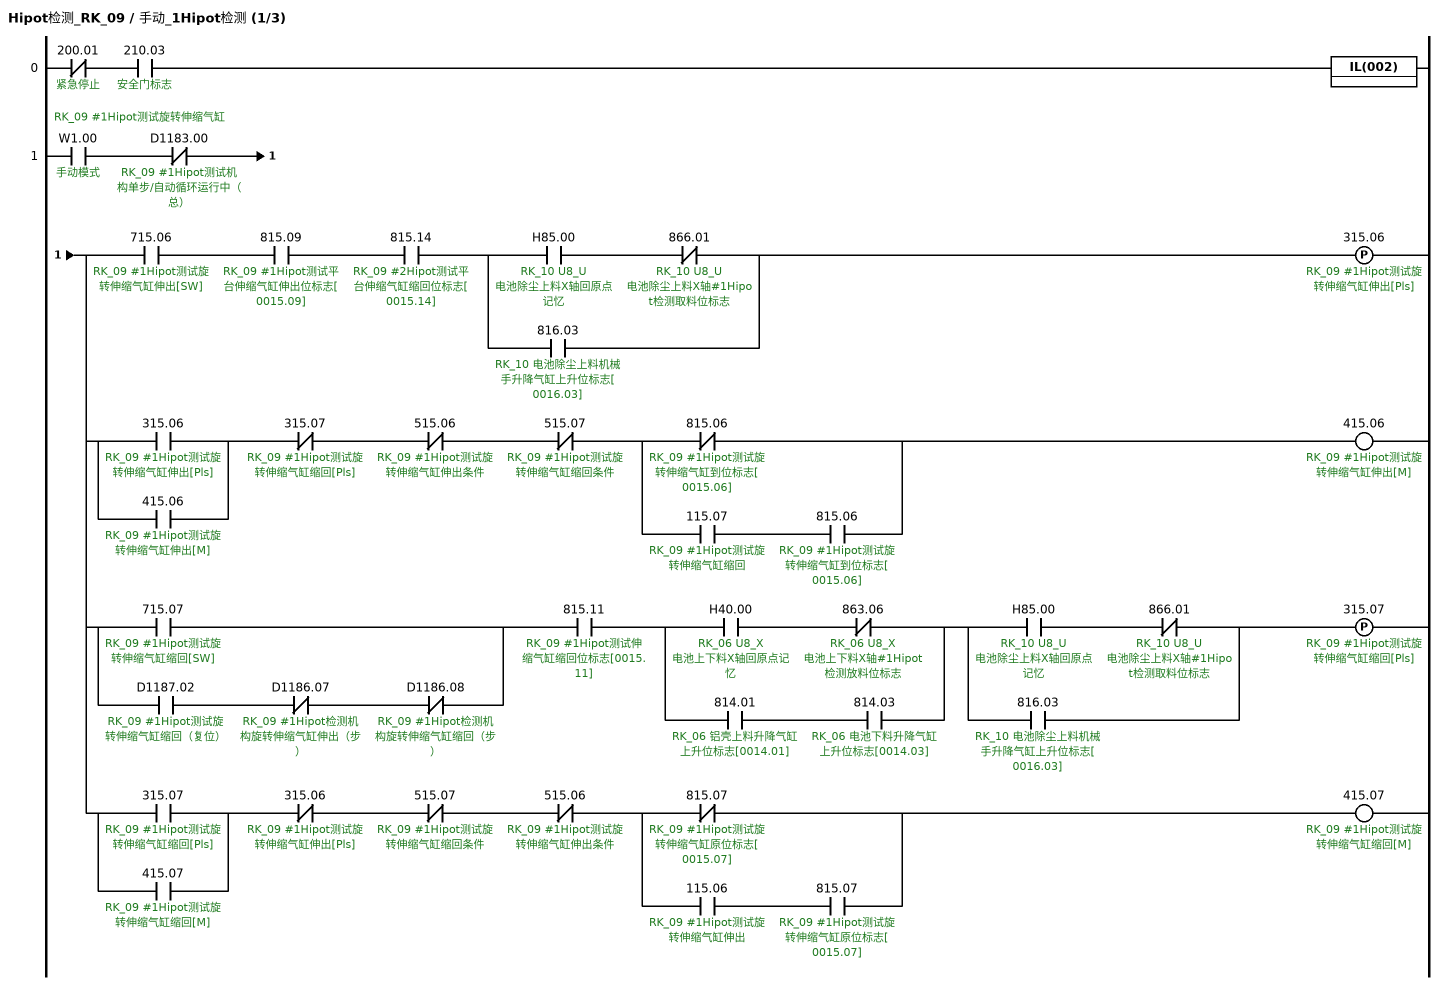
; [picture p648: Hipot检测_RK_09 / 手动_1Hipot检测, rungs 0-1]
; rung 0
LDNOT 200.01  ; 紧急停止
AND 210.03  ; 安全门标志
IL(002)
; rung 1: RK_09 #1Hipot测试旋转伸缩气缸
LD W1.00  ; 手动模式
ANDNOT D1183.00  ; RK_09 #1Hipot测试机构单步/自动循环运行中（总）
OUT TR0
AND 715.06  ; RK_09 #1Hipot测试旋转伸缩气缸伸出[SW]
AND 815.09  ; RK_09 #1Hipot测试平台伸缩气缸伸出位标志[0015.09]
AND 815.14  ; RK_09 #2Hipot测试平台伸缩气缸缩回位标志[0015.14]
LD H85.00  ; RK_10 U8_U 电池除尘上料X轴回原点记忆
ANDNOT 866.01  ; RK_10 U8_U 电池除尘上料X轴#1Hipot检测取料位标志
OR 816.03  ; RK_10 电池除尘上料机械手升降气缸上升位标志[0016.03]
ANDLD
DIFU(013) 315.06  ; RK_09 #1Hipot测试旋转伸缩气缸伸出[Pls]
LD TR0
LD 315.06  ; RK_09 #1Hipot测试旋转伸缩气缸伸出[Pls]
OR 415.06  ; RK_09 #1Hipot测试旋转伸缩气缸伸出[M]
ANDLD
ANDNOT 315.07  ; RK_09 #1Hipot测试旋转伸缩气缸缩回[Pls]
ANDNOT 515.06  ; RK_09 #1Hipot测试旋转伸缩气缸伸出条件
ANDNOT 515.07  ; RK_09 #1Hipot测试旋转伸缩气缸缩回条件
LDNOT 815.06  ; RK_09 #1Hipot测试旋转伸缩气缸到位标志[0015.06]
LD 115.07  ; RK_09 #1Hipot测试旋转伸缩气缸缩回
AND 815.06  ; RK_09 #1Hipot测试旋转伸缩气缸到位标志[0015.06]
ORLD
ANDLD
OUT 415.06  ; RK_09 #1Hipot测试旋转伸缩气缸伸出[M]
LD TR0
LD 715.07  ; RK_09 #1Hipot测试旋转伸缩气缸缩回[SW]
LD D1187.02  ; RK_09 #1Hipot测试旋转伸缩气缸缩回（复位）
ANDNOT D1186.07  ; RK_09 #1Hipot检测机构旋转伸缩气缸伸出（步）
ANDNOT D1186.08  ; RK_09 #1Hipot检测机构旋转伸缩气缸缩回（步）
ORLD
ANDLD
AND 815.11  ; RK_09 #1Hipot测试伸缩气缸缩回位标志[0015.11]
LD H40.00  ; RK_06 U8_X 电池上下料X轴回原点记忆
ANDNOT 863.06  ; RK_06 U8_X 电池上下料X轴#1Hipot检测放料位标志
LD 814.01  ; RK_06 铝壳上料升降气缸上升位标志[0014.01]
AND 814.03  ; RK_06 电池下料升降气缸上升位标志[0014.03]
ORLD
ANDLD
LD H85.00  ; RK_10 U8_U 电池除尘上料X轴回原点记忆
ANDNOT 866.01  ; RK_10 U8_U 电池除尘上料X轴#1Hipot检测取料位标志
OR 816.03  ; RK_10 电池除尘上料机械手升降气缸上升位标志[0016.03]
ANDLD
DIFU(013) 315.07  ; RK_09 #1Hipot测试旋转伸缩气缸缩回[Pls]
LD TR0
LD 315.07  ; RK_09 #1Hipot测试旋转伸缩气缸缩回[Pls]
OR 415.07  ; RK_09 #1Hipot测试旋转伸缩气缸缩回[M]
ANDLD
ANDNOT 315.06  ; RK_09 #1Hipot测试旋转伸缩气缸伸出[Pls]
ANDNOT 515.07  ; RK_09 #1Hipot测试旋转伸缩气缸缩回条件
ANDNOT 515.06  ; RK_09 #1Hipot测试旋转伸缩气缸伸出条件
LDNOT 815.07  ; RK_09 #1Hipot测试旋转伸缩气缸原位标志[0015.07]
LD 115.06  ; RK_09 #1Hipot测试旋转伸缩气缸伸出
AND 815.07  ; RK_09 #1Hipot测试旋转伸缩气缸原位标志[0015.07]
ORLD
ANDLD
OUT 415.07  ; RK_09 #1Hipot测试旋转伸缩气缸缩回[M]

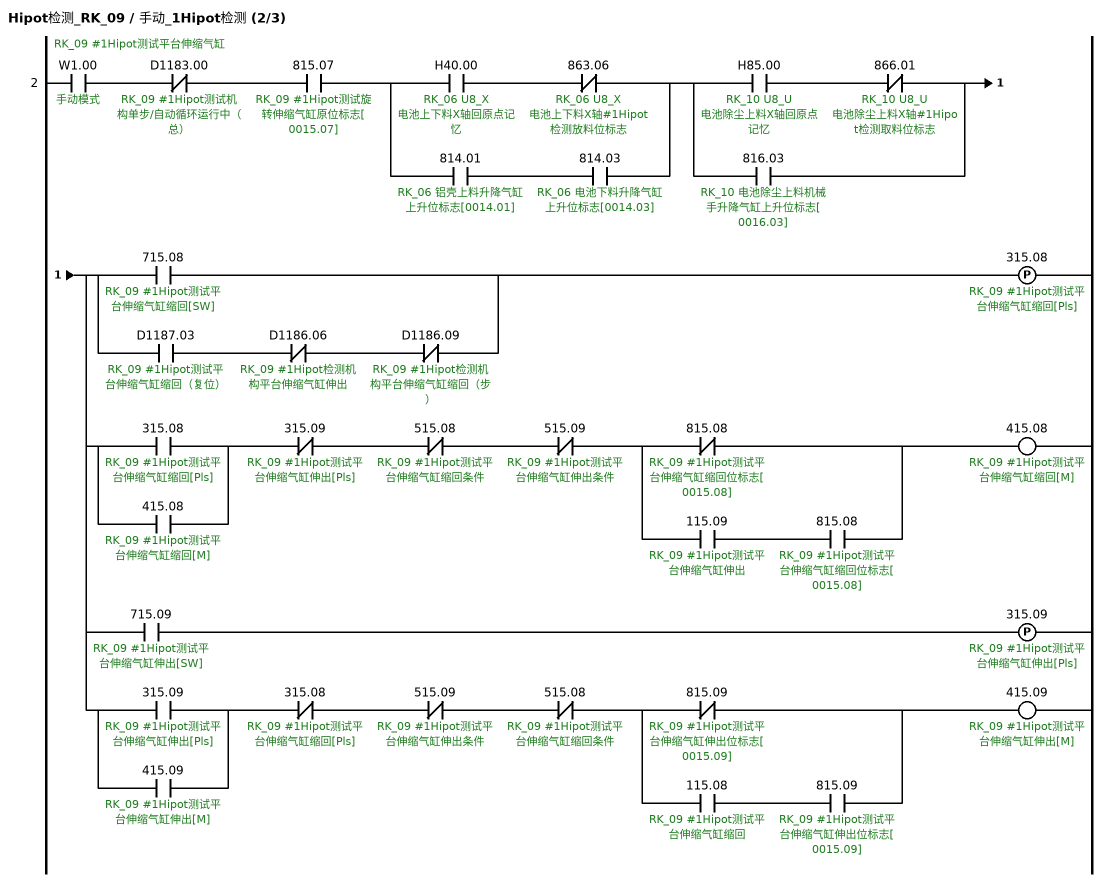
; rung 2: RK_09 #1Hipot测试平台伸缩气缸
LD W1.00  ; 手动模式
ANDNOT D1183.00  ; RK_09 #1Hipot测试机构单步/自动循环运行中（总）
AND 815.07  ; RK_09 #1Hipot测试旋转伸缩气缸原位标志[0015.07]
LD H40.00  ; RK_06 U8_X 电池上下料X轴回原点记忆
ANDNOT 863.06  ; RK_06 U8_X 电池上下料X轴#1Hipot检测放料位标志
LD 814.01  ; RK_06 铝壳上料升降气缸上升位标志[0014.01]
AND 814.03  ; RK_06 电池下料升降气缸上升位标志[0014.03]
ORLD
ANDLD
LD H85.00  ; RK_10 U8_U 电池除尘上料X轴回原点记忆
ANDNOT 866.01  ; RK_10 U8_U 电池除尘上料X轴#1Hipot检测取料位标志
OR 816.03  ; RK_10 电池除尘上料机械手升降气缸上升位标志[0016.03]
ANDLD
OUT TR0
LD 715.08  ; RK_09 #1Hipot测试平台伸缩气缸缩回[SW]
LD D1187.03  ; RK_09 #1Hipot测试平台伸缩气缸缩回（复位）
ANDNOT D1186.06  ; RK_09 #1Hipot检测机构平台伸缩气缸伸出
ANDNOT D1186.09  ; RK_09 #1Hipot检测机构平台伸缩气缸缩回（步）
ORLD
ANDLD
DIFU(013) 315.08  ; RK_09 #1Hipot测试平台伸缩气缸缩回[Pls]
LD TR0
LD 315.08  ; RK_09 #1Hipot测试平台伸缩气缸缩回[Pls]
OR 415.08  ; RK_09 #1Hipot测试平台伸缩气缸缩回[M]
ANDLD
ANDNOT 315.09  ; RK_09 #1Hipot测试平台伸缩气缸伸出[Pls]
ANDNOT 515.08  ; RK_09 #1Hipot测试平台伸缩气缸缩回条件
ANDNOT 515.09  ; RK_09 #1Hipot测试平台伸缩气缸伸出条件
LDNOT 815.08  ; RK_09 #1Hipot测试平台伸缩气缸缩回位标志[0015.08]
LD 115.09  ; RK_09 #1Hipot测试平台伸缩气缸伸出
AND 815.08  ; RK_09 #1Hipot测试平台伸缩气缸缩回位标志[0015.08]
ORLD
ANDLD
OUT 415.08  ; RK_09 #1Hipot测试平台伸缩气缸缩回[M]
LD TR0
AND 715.09  ; RK_09 #1Hipot测试平台伸缩气缸伸出[SW]
DIFU(013) 315.09  ; RK_09 #1Hipot测试平台伸缩气缸伸出[Pls]
LD TR0
LD 315.09  ; RK_09 #1Hipot测试平台伸缩气缸伸出[Pls]
OR 415.09  ; RK_09 #1Hipot测试平台伸缩气缸伸出[M]
ANDLD
ANDNOT 315.08  ; RK_09 #1Hipot测试平台伸缩气缸缩回[Pls]
ANDNOT 515.09  ; RK_09 #1Hipot测试平台伸缩气缸伸出条件
ANDNOT 515.08  ; RK_09 #1Hipot测试平台伸缩气缸缩回条件
LDNOT 815.09  ; RK_09 #1Hipot测试平台伸缩气缸伸出位标志[0015.09]
LD 115.08  ; RK_09 #1Hipot测试平台伸缩气缸缩回
AND 815.09  ; RK_09 #1Hipot测试平台伸缩气缸伸出位标志[0015.09]
ORLD
ANDLD
OUT 415.09  ; RK_09 #1Hipot测试平台伸缩气缸伸出[M]

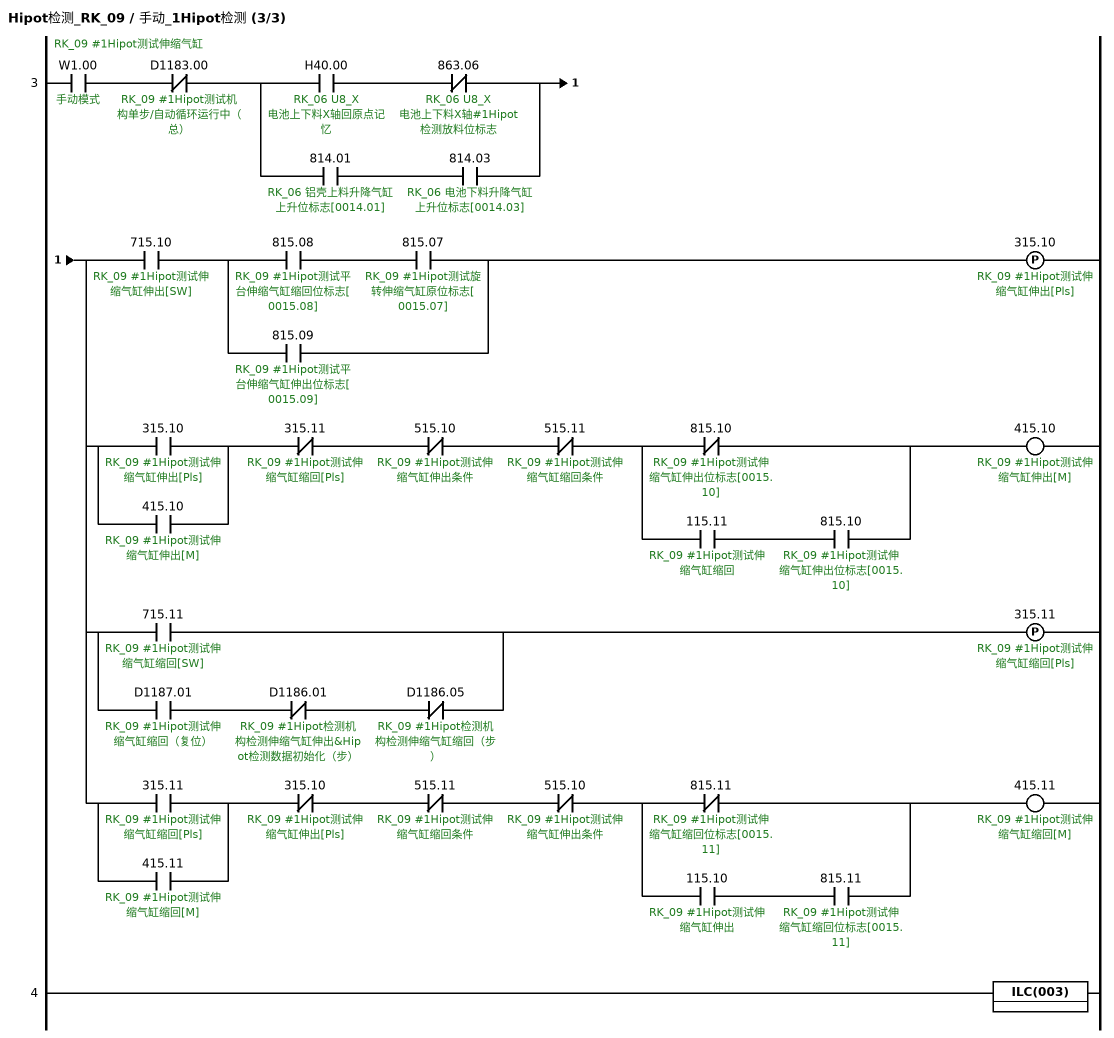
; rung 3: RK_09 #1Hipot测试伸缩气缸
LD W1.00  ; 手动模式
ANDNOT D1183.00  ; RK_09 #1Hipot测试机构单步/自动循环运行中（总）
LD H40.00  ; RK_06 U8_X 电池上下料X轴回原点记忆
ANDNOT 863.06  ; RK_06 U8_X 电池上下料X轴#1Hipot检测放料位标志
LD 814.01  ; RK_06 铝壳上料升降气缸上升位标志[0014.01]
AND 814.03  ; RK_06 电池下料升降气缸上升位标志[0014.03]
ORLD
ANDLD
OUT TR0
AND 715.10  ; RK_09 #1Hipot测试伸缩气缸伸出[SW]
LD 815.08  ; RK_09 #1Hipot测试平台伸缩气缸缩回位标志[0015.08]
AND 815.07  ; RK_09 #1Hipot测试旋转伸缩气缸原位标志[0015.07]
OR 815.09  ; RK_09 #1Hipot测试平台伸缩气缸伸出位标志[0015.09]
ANDLD
DIFU(013) 315.10  ; RK_09 #1Hipot测试伸缩气缸伸出[Pls]
LD TR0
LD 315.10  ; RK_09 #1Hipot测试伸缩气缸伸出[Pls]
OR 415.10  ; RK_09 #1Hipot测试伸缩气缸伸出[M]
ANDLD
ANDNOT 315.11  ; RK_09 #1Hipot测试伸缩气缸缩回[Pls]
ANDNOT 515.10  ; RK_09 #1Hipot测试伸缩气缸伸出条件
ANDNOT 515.11  ; RK_09 #1Hipot测试伸缩气缸缩回条件
LDNOT 815.10  ; RK_09 #1Hipot测试伸缩气缸伸出位标志[0015.10]
LD 115.11  ; RK_09 #1Hipot测试伸缩气缸缩回
AND 815.10  ; RK_09 #1Hipot测试伸缩气缸伸出位标志[0015.10]
ORLD
ANDLD
OUT 415.10  ; RK_09 #1Hipot测试伸缩气缸伸出[M]
LD TR0
LD 715.11  ; RK_09 #1Hipot测试伸缩气缸缩回[SW]
LD D1187.01  ; RK_09 #1Hipot测试伸缩气缸缩回（复位）
ANDNOT D1186.01  ; RK_09 #1Hipot检测机构检测伸缩气缸伸出&Hipot检测数据初始化（步）
ANDNOT D1186.05  ; RK_09 #1Hipot检测机构检测伸缩气缸缩回（步）
ORLD
ANDLD
DIFU(013) 315.11  ; RK_09 #1Hipot测试伸缩气缸缩回[Pls]
LD TR0
LD 315.11  ; RK_09 #1Hipot测试伸缩气缸缩回[Pls]
OR 415.11  ; RK_09 #1Hipot测试伸缩气缸缩回[M]
ANDLD
ANDNOT 315.10  ; RK_09 #1Hipot测试伸缩气缸伸出[Pls]
ANDNOT 515.11  ; RK_09 #1Hipot测试伸缩气缸缩回条件
ANDNOT 515.10  ; RK_09 #1Hipot测试伸缩气缸伸出条件
LDNOT 815.11  ; RK_09 #1Hipot测试伸缩气缸缩回位标志[0015.11]
LD 115.10  ; RK_09 #1Hipot测试伸缩气缸伸出
AND 815.11  ; RK_09 #1Hipot测试伸缩气缸缩回位标志[0015.11]
ORLD
ANDLD
OUT 415.11  ; RK_09 #1Hipot测试伸缩气缸缩回[M]
; rung 4
ILC(003)

### Section 手动_2Hipot检测

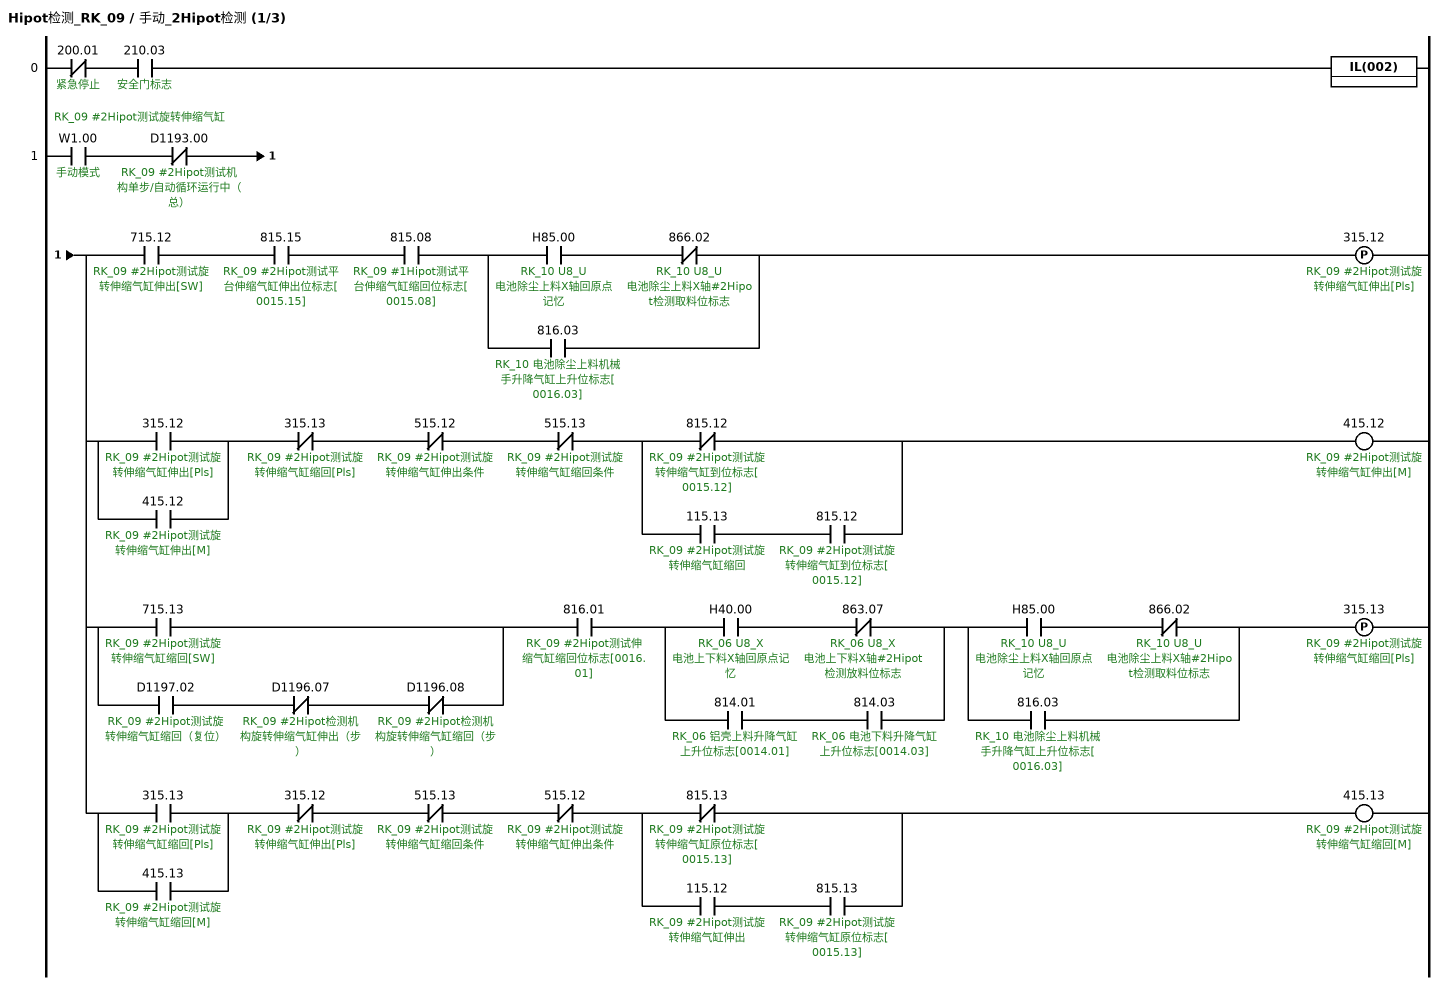
; rung 0
LDNOT 200.01  ; 紧急停止
AND 210.03  ; 安全门标志
IL(002)
; rung 1: RK_09 #2Hipot测试旋转伸缩气缸
LD W1.00  ; 手动模式
ANDNOT D1193.00  ; RK_09 #2Hipot测试机构单步/自动循环运行中（总）
OUT TR0
AND 715.12  ; RK_09 #2Hipot测试旋转伸缩气缸伸出[SW]
AND 815.15  ; RK_09 #2Hipot测试平台伸缩气缸伸出位标志[0015.15]
AND 815.08  ; RK_09 #1Hipot测试平台伸缩气缸缩回位标志[0015.08]
LD H85.00  ; RK_10 U8_U 电池除尘上料X轴回原点记忆
ANDNOT 866.02  ; RK_10 U8_U 电池除尘上料X轴#2Hipot检测取料位标志
OR 816.03  ; RK_10 电池除尘上料机械手升降气缸上升位标志[0016.03]
ANDLD
DIFU(013) 315.12  ; RK_09 #2Hipot测试旋转伸缩气缸伸出[Pls]
LD TR0
LD 315.12  ; RK_09 #2Hipot测试旋转伸缩气缸伸出[Pls]
OR 415.12  ; RK_09 #2Hipot测试旋转伸缩气缸伸出[M]
ANDLD
ANDNOT 315.13  ; RK_09 #2Hipot测试旋转伸缩气缸缩回[Pls]
ANDNOT 515.12  ; RK_09 #2Hipot测试旋转伸缩气缸伸出条件
ANDNOT 515.13  ; RK_09 #2Hipot测试旋转伸缩气缸缩回条件
LDNOT 815.12  ; RK_09 #2Hipot测试旋转伸缩气缸到位标志[0015.12]
LD 115.13  ; RK_09 #2Hipot测试旋转伸缩气缸缩回
AND 815.12  ; RK_09 #2Hipot测试旋转伸缩气缸到位标志[0015.12]
ORLD
ANDLD
OUT 415.12  ; RK_09 #2Hipot测试旋转伸缩气缸伸出[M]
LD TR0
LD 715.13  ; RK_09 #2Hipot测试旋转伸缩气缸缩回[SW]
LD D1197.02  ; RK_09 #2Hipot测试旋转伸缩气缸缩回（复位）
ANDNOT D1196.07  ; RK_09 #2Hipot检测机构旋转伸缩气缸伸出（步）
ANDNOT D1196.08  ; RK_09 #2Hipot检测机构旋转伸缩气缸缩回（步）
ORLD
ANDLD
AND 816.01  ; RK_09 #2Hipot测试伸缩气缸缩回位标志[0016.01]
LD H40.00  ; RK_06 U8_X 电池上下料X轴回原点记忆
ANDNOT 863.07  ; RK_06 U8_X 电池上下料X轴#2Hipot检测放料位标志
LD 814.01  ; RK_06 铝壳上料升降气缸上升位标志[0014.01]
AND 814.03  ; RK_06 电池下料升降气缸上升位标志[0014.03]
ORLD
ANDLD
LD H85.00  ; RK_10 U8_U 电池除尘上料X轴回原点记忆
ANDNOT 866.02  ; RK_10 U8_U 电池除尘上料X轴#2Hipot检测取料位标志
OR 816.03  ; RK_10 电池除尘上料机械手升降气缸上升位标志[0016.03]
ANDLD
DIFU(013) 315.13  ; RK_09 #2Hipot测试旋转伸缩气缸缩回[Pls]
LD TR0
LD 315.13  ; RK_09 #2Hipot测试旋转伸缩气缸缩回[Pls]
OR 415.13  ; RK_09 #2Hipot测试旋转伸缩气缸缩回[M]
ANDLD
ANDNOT 315.12  ; RK_09 #2Hipot测试旋转伸缩气缸伸出[Pls]
ANDNOT 515.13  ; RK_09 #2Hipot测试旋转伸缩气缸缩回条件
ANDNOT 515.12  ; RK_09 #2Hipot测试旋转伸缩气缸伸出条件
LDNOT 815.13  ; RK_09 #2Hipot测试旋转伸缩气缸原位标志[0015.13]
LD 115.12  ; RK_09 #2Hipot测试旋转伸缩气缸伸出
AND 815.13  ; RK_09 #2Hipot测试旋转伸缩气缸原位标志[0015.13]
ORLD
ANDLD
OUT 415.13  ; RK_09 #2Hipot测试旋转伸缩气缸缩回[M]

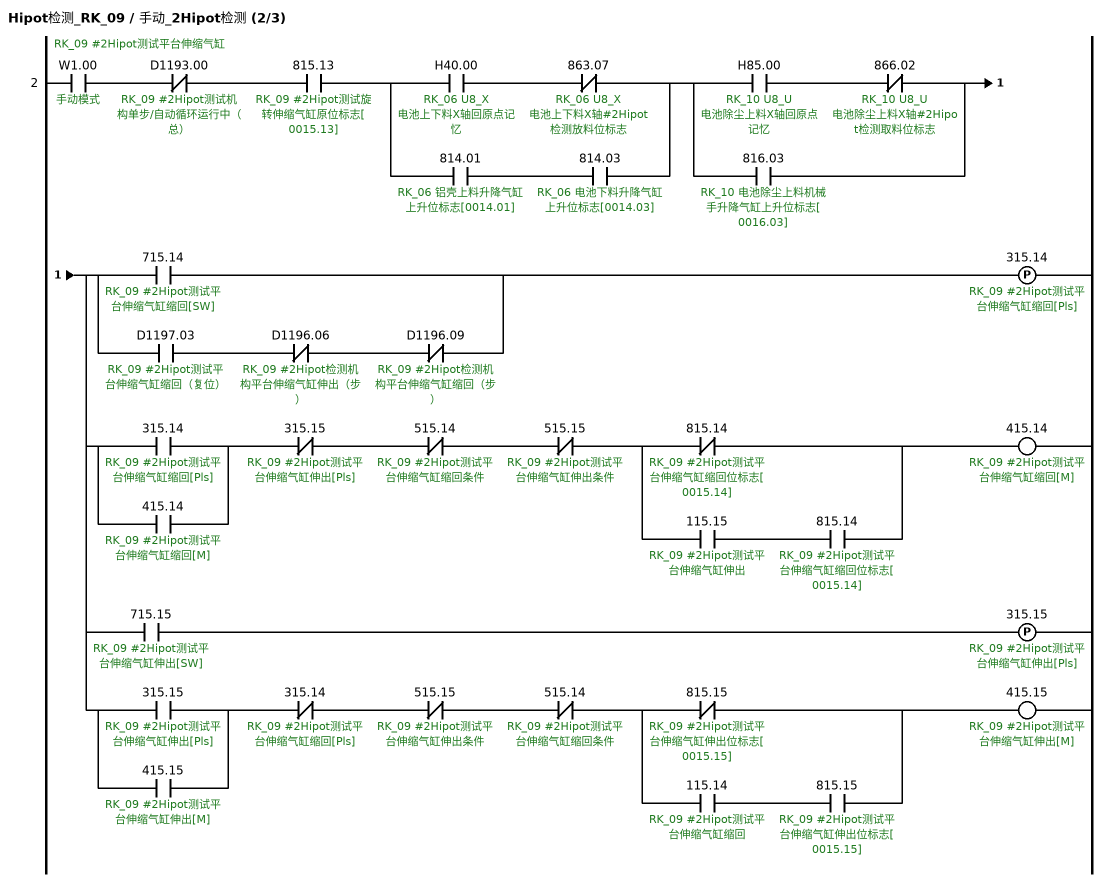
; rung 2: RK_09 #2Hipot测试平台伸缩气缸
LD W1.00  ; 手动模式
ANDNOT D1193.00  ; RK_09 #2Hipot测试机构单步/自动循环运行中（总）
AND 815.13  ; RK_09 #2Hipot测试旋转伸缩气缸原位标志[0015.13]
LD H40.00  ; RK_06 U8_X 电池上下料X轴回原点记忆
ANDNOT 863.07  ; RK_06 U8_X 电池上下料X轴#2Hipot检测放料位标志
LD 814.01  ; RK_06 铝壳上料升降气缸上升位标志[0014.01]
AND 814.03  ; RK_06 电池下料升降气缸上升位标志[0014.03]
ORLD
ANDLD
LD H85.00  ; RK_10 U8_U 电池除尘上料X轴回原点记忆
ANDNOT 866.02  ; RK_10 U8_U 电池除尘上料X轴#2Hipot检测取料位标志
OR 816.03  ; RK_10 电池除尘上料机械手升降气缸上升位标志[0016.03]
ANDLD
OUT TR0
LD 715.14  ; RK_09 #2Hipot测试平台伸缩气缸缩回[SW]
LD D1197.03  ; RK_09 #2Hipot测试平台伸缩气缸缩回（复位）
ANDNOT D1196.06  ; RK_09 #2Hipot检测机构平台伸缩气缸伸出（步）
ANDNOT D1196.09  ; RK_09 #2Hipot检测机构平台伸缩气缸缩回（步）
ORLD
ANDLD
DIFU(013) 315.14  ; RK_09 #2Hipot测试平台伸缩气缸缩回[Pls]
LD TR0
LD 315.14  ; RK_09 #2Hipot测试平台伸缩气缸缩回[Pls]
OR 415.14  ; RK_09 #2Hipot测试平台伸缩气缸缩回[M]
ANDLD
ANDNOT 315.15  ; RK_09 #2Hipot测试平台伸缩气缸伸出[Pls]
ANDNOT 515.14  ; RK_09 #2Hipot测试平台伸缩气缸缩回条件
ANDNOT 515.15  ; RK_09 #2Hipot测试平台伸缩气缸伸出条件
LDNOT 815.14  ; RK_09 #2Hipot测试平台伸缩气缸缩回位标志[0015.14]
LD 115.15  ; RK_09 #2Hipot测试平台伸缩气缸伸出
AND 815.14  ; RK_09 #2Hipot测试平台伸缩气缸缩回位标志[0015.14]
ORLD
ANDLD
OUT 415.14  ; RK_09 #2Hipot测试平台伸缩气缸缩回[M]
LD TR0
AND 715.15  ; RK_09 #2Hipot测试平台伸缩气缸伸出[SW]
DIFU(013) 315.15  ; RK_09 #2Hipot测试平台伸缩气缸伸出[Pls]
LD TR0
LD 315.15  ; RK_09 #2Hipot测试平台伸缩气缸伸出[Pls]
OR 415.15  ; RK_09 #2Hipot测试平台伸缩气缸伸出[M]
ANDLD
ANDNOT 315.14  ; RK_09 #2Hipot测试平台伸缩气缸缩回[Pls]
ANDNOT 515.15  ; RK_09 #2Hipot测试平台伸缩气缸伸出条件
ANDNOT 515.14  ; RK_09 #2Hipot测试平台伸缩气缸缩回条件
LDNOT 815.15  ; RK_09 #2Hipot测试平台伸缩气缸伸出位标志[0015.15]
LD 115.14  ; RK_09 #2Hipot测试平台伸缩气缸缩回
AND 815.15  ; RK_09 #2Hipot测试平台伸缩气缸伸出位标志[0015.15]
ORLD
ANDLD
OUT 415.15  ; RK_09 #2Hipot测试平台伸缩气缸伸出[M]

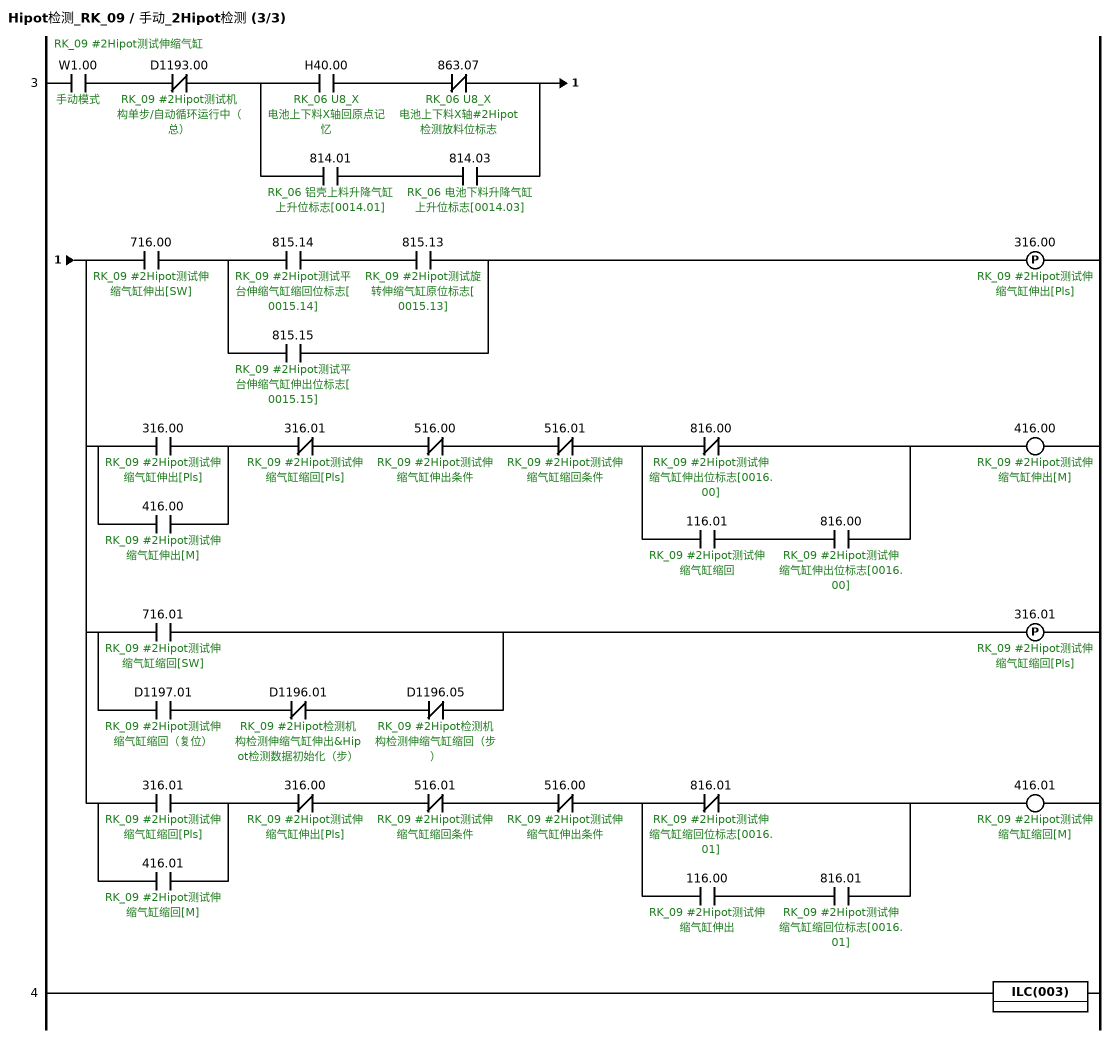
; rung 3: RK_09 #2Hipot测试伸缩气缸
LD W1.00  ; 手动模式
ANDNOT D1193.00  ; RK_09 #2Hipot测试机构单步/自动循环运行中（总）
LD H40.00  ; RK_06 U8_X 电池上下料X轴回原点记忆
ANDNOT 863.07  ; RK_06 U8_X 电池上下料X轴#2Hipot检测放料位标志
LD 814.01  ; RK_06 铝壳上料升降气缸上升位标志[0014.01]
AND 814.03  ; RK_06 电池下料升降气缸上升位标志[0014.03]
ORLD
ANDLD
OUT TR0
AND 716.00  ; RK_09 #2Hipot测试伸缩气缸伸出[SW]
LD 815.14  ; RK_09 #2Hipot测试平台伸缩气缸缩回位标志[0015.14]
AND 815.13  ; RK_09 #2Hipot测试旋转伸缩气缸原位标志[0015.13]
OR 815.15  ; RK_09 #2Hipot测试平台伸缩气缸伸出位标志[0015.15]
ANDLD
DIFU(013) 316.00  ; RK_09 #2Hipot测试伸缩气缸伸出[Pls]
LD TR0
LD 316.00  ; RK_09 #2Hipot测试伸缩气缸伸出[Pls]
OR 416.00  ; RK_09 #2Hipot测试伸缩气缸伸出[M]
ANDLD
ANDNOT 316.01  ; RK_09 #2Hipot测试伸缩气缸缩回[Pls]
ANDNOT 516.00  ; RK_09 #2Hipot测试伸缩气缸伸出条件
ANDNOT 516.01  ; RK_09 #2Hipot测试伸缩气缸缩回条件
LDNOT 816.00  ; RK_09 #2Hipot测试伸缩气缸伸出位标志[0016.00]
LD 116.01  ; RK_09 #2Hipot测试伸缩气缸缩回
AND 816.00  ; RK_09 #2Hipot测试伸缩气缸伸出位标志[0016.00]
ORLD
ANDLD
OUT 416.00  ; RK_09 #2Hipot测试伸缩气缸伸出[M]
LD TR0
LD 716.01  ; RK_09 #2Hipot测试伸缩气缸缩回[SW]
LD D1197.01  ; RK_09 #2Hipot测试伸缩气缸缩回（复位）
ANDNOT D1196.01  ; RK_09 #2Hipot检测机构检测伸缩气缸伸出&Hipot检测数据初始化（步）
ANDNOT D1196.05  ; RK_09 #2Hipot检测机构检测伸缩气缸缩回（步）
ORLD
ANDLD
DIFU(013) 316.01  ; RK_09 #2Hipot测试伸缩气缸缩回[Pls]
LD TR0
LD 316.01  ; RK_09 #2Hipot测试伸缩气缸缩回[Pls]
OR 416.01  ; RK_09 #2Hipot测试伸缩气缸缩回[M]
ANDLD
ANDNOT 316.00  ; RK_09 #2Hipot测试伸缩气缸伸出[Pls]
ANDNOT 516.01  ; RK_09 #2Hipot测试伸缩气缸缩回条件
ANDNOT 516.00  ; RK_09 #2Hipot测试伸缩气缸伸出条件
LDNOT 816.01  ; RK_09 #2Hipot测试伸缩气缸缩回位标志[0016.01]
LD 116.00  ; RK_09 #2Hipot测试伸缩气缸伸出
AND 816.01  ; RK_09 #2Hipot测试伸缩气缸缩回位标志[0016.01]
ORLD
ANDLD
OUT 416.01  ; RK_09 #2Hipot测试伸缩气缸缩回[M]
; rung 4
ILC(003)

### Section 自动_1Hipot检测

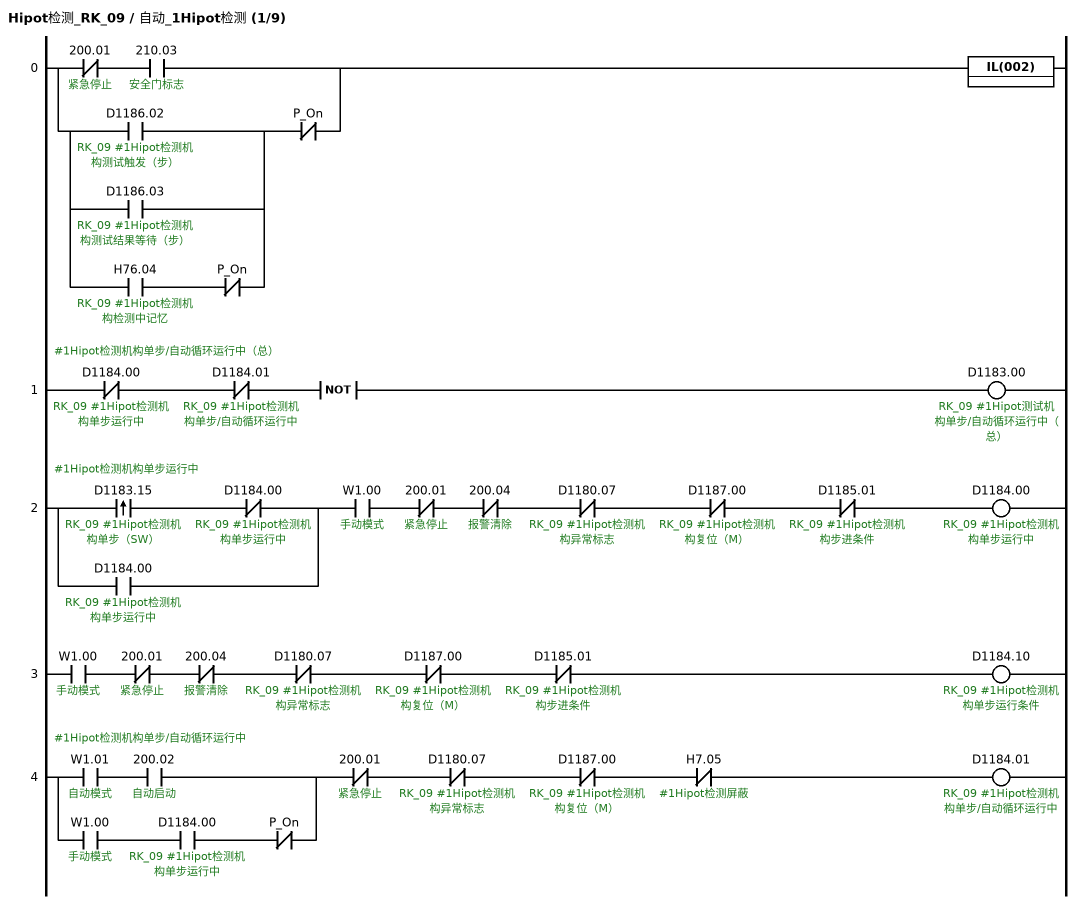
; rung 0
LDNOT 200.01  ; 紧急停止
AND 210.03  ; 安全门标志
LD D1186.02  ; RK_09 #1Hipot检测机构测试触发（步）
OR D1186.03  ; RK_09 #1Hipot检测机构测试结果等待（步）
LD H76.04  ; RK_09 #1Hipot检测机构检测中记忆
ANDNOT P_On
ORLD
ANDNOT P_On  // Hipot测试触发后，急停|安全门打开情况下测试继续，直到有测试完成信号！
ORLD
IL(002)
; rung 1: #1Hipot检测机构单步/自动循环运行中（总）
LDNOT D1184.00  ; RK_09 #1Hipot检测机构单步运行中
ANDNOT D1184.01  ; RK_09 #1Hipot检测机构单步/自动循环运行中
NOT(520)
OUT D1183.00  ; RK_09 #1Hipot测试机构单步/自动循环运行中（总）
; rung 2: #1Hipot检测机构单步运行中
@LD D1183.15  ; RK_09 #1Hipot检测机构单步（SW）
ANDNOT D1184.00  ; RK_09 #1Hipot检测机构单步运行中
OR D1184.00  ; RK_09 #1Hipot检测机构单步运行中
AND W1.00  ; 手动模式
ANDNOT 200.01  ; 紧急停止
ANDNOT 200.04  ; 报警清除
ANDNOT D1180.07  ; RK_09 #1Hipot检测机构异常标志
ANDNOT D1187.00  ; RK_09 #1Hipot检测机构复位（M）
ANDNOT D1185.01  ; RK_09 #1Hipot检测机构步进条件
OUT D1184.00  ; RK_09 #1Hipot检测机构单步运行中
; rung 3
LD W1.00  ; 手动模式
ANDNOT 200.01  ; 紧急停止
ANDNOT 200.04  ; 报警清除
ANDNOT D1180.07  ; RK_09 #1Hipot检测机构异常标志
ANDNOT D1187.00  ; RK_09 #1Hipot检测机构复位（M）
ANDNOT D1185.01  ; RK_09 #1Hipot检测机构步进条件
OUT D1184.10  ; RK_09 #1Hipot检测机构单步运行条件
; rung 4: #1Hipot检测机构单步/自动循环运行中
LD W1.01  ; 自动模式
AND 200.02  ; 自动启动
LD W1.00  ; 手动模式
AND D1184.00  ; RK_09 #1Hipot检测机构单步运行中
ANDNOT P_On
ORLD
ANDNOT 200.01  ; 紧急停止
ANDNOT D1180.07  ; RK_09 #1Hipot检测机构异常标志
ANDNOT D1187.00  ; RK_09 #1Hipot检测机构复位（M）
ANDNOT H7.05  ; #1Hipot检测屏蔽
OUT D1184.01  ; RK_09 #1Hipot检测机构单步/自动循环运行中

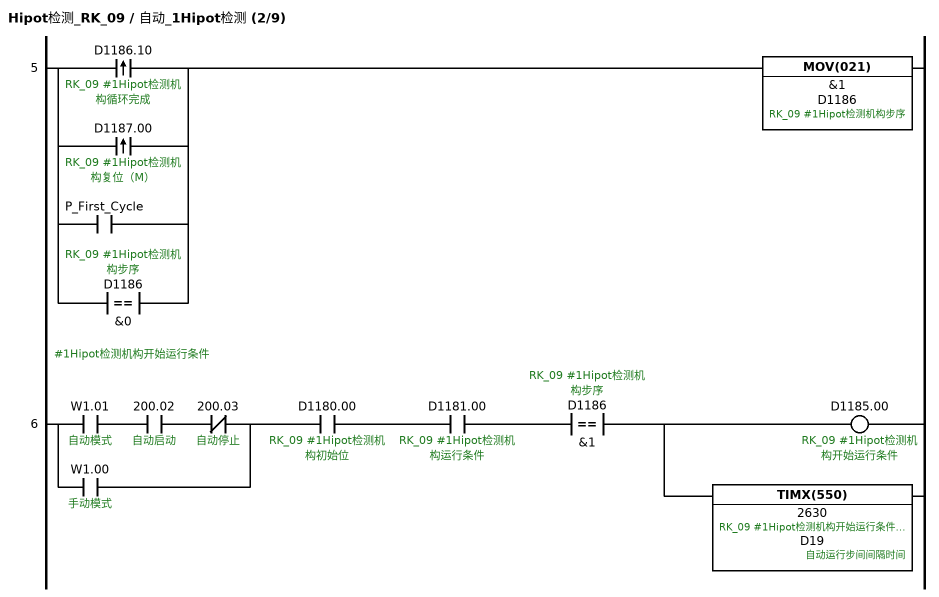
; rung 5
@LD D1186.10  ; RK_09 #1Hipot检测机构循环完成
@OR D1187.00  ; RK_09 #1Hipot检测机构复位（M）
OR P_First_Cycle
OR=(300) D1186 &0  ; RK_09 #1Hipot检测机构步序
MOV(021) &1 D1186  ; RK_09 #1Hipot检测机构步序
; rung 6: #1Hipot检测机构开始运行条件
LD W1.01  ; 自动模式
AND 200.02  ; 自动启动
ANDNOT 200.03  ; 自动停止
OR W1.00  ; 手动模式
AND D1180.00  ; RK_09 #1Hipot检测机构初始位
AND D1181.00  ; RK_09 #1Hipot检测机构运行条件
AND=(300) D1186 &1  ; RK_09 #1Hipot检测机构步序
OUT D1185.00  ; RK_09 #1Hipot检测机构开始运行条件
TIMX(550) 2630 D19  ; 自动运行步间间隔时间, RK_09 #1Hipot检测机构开始运行条件延时

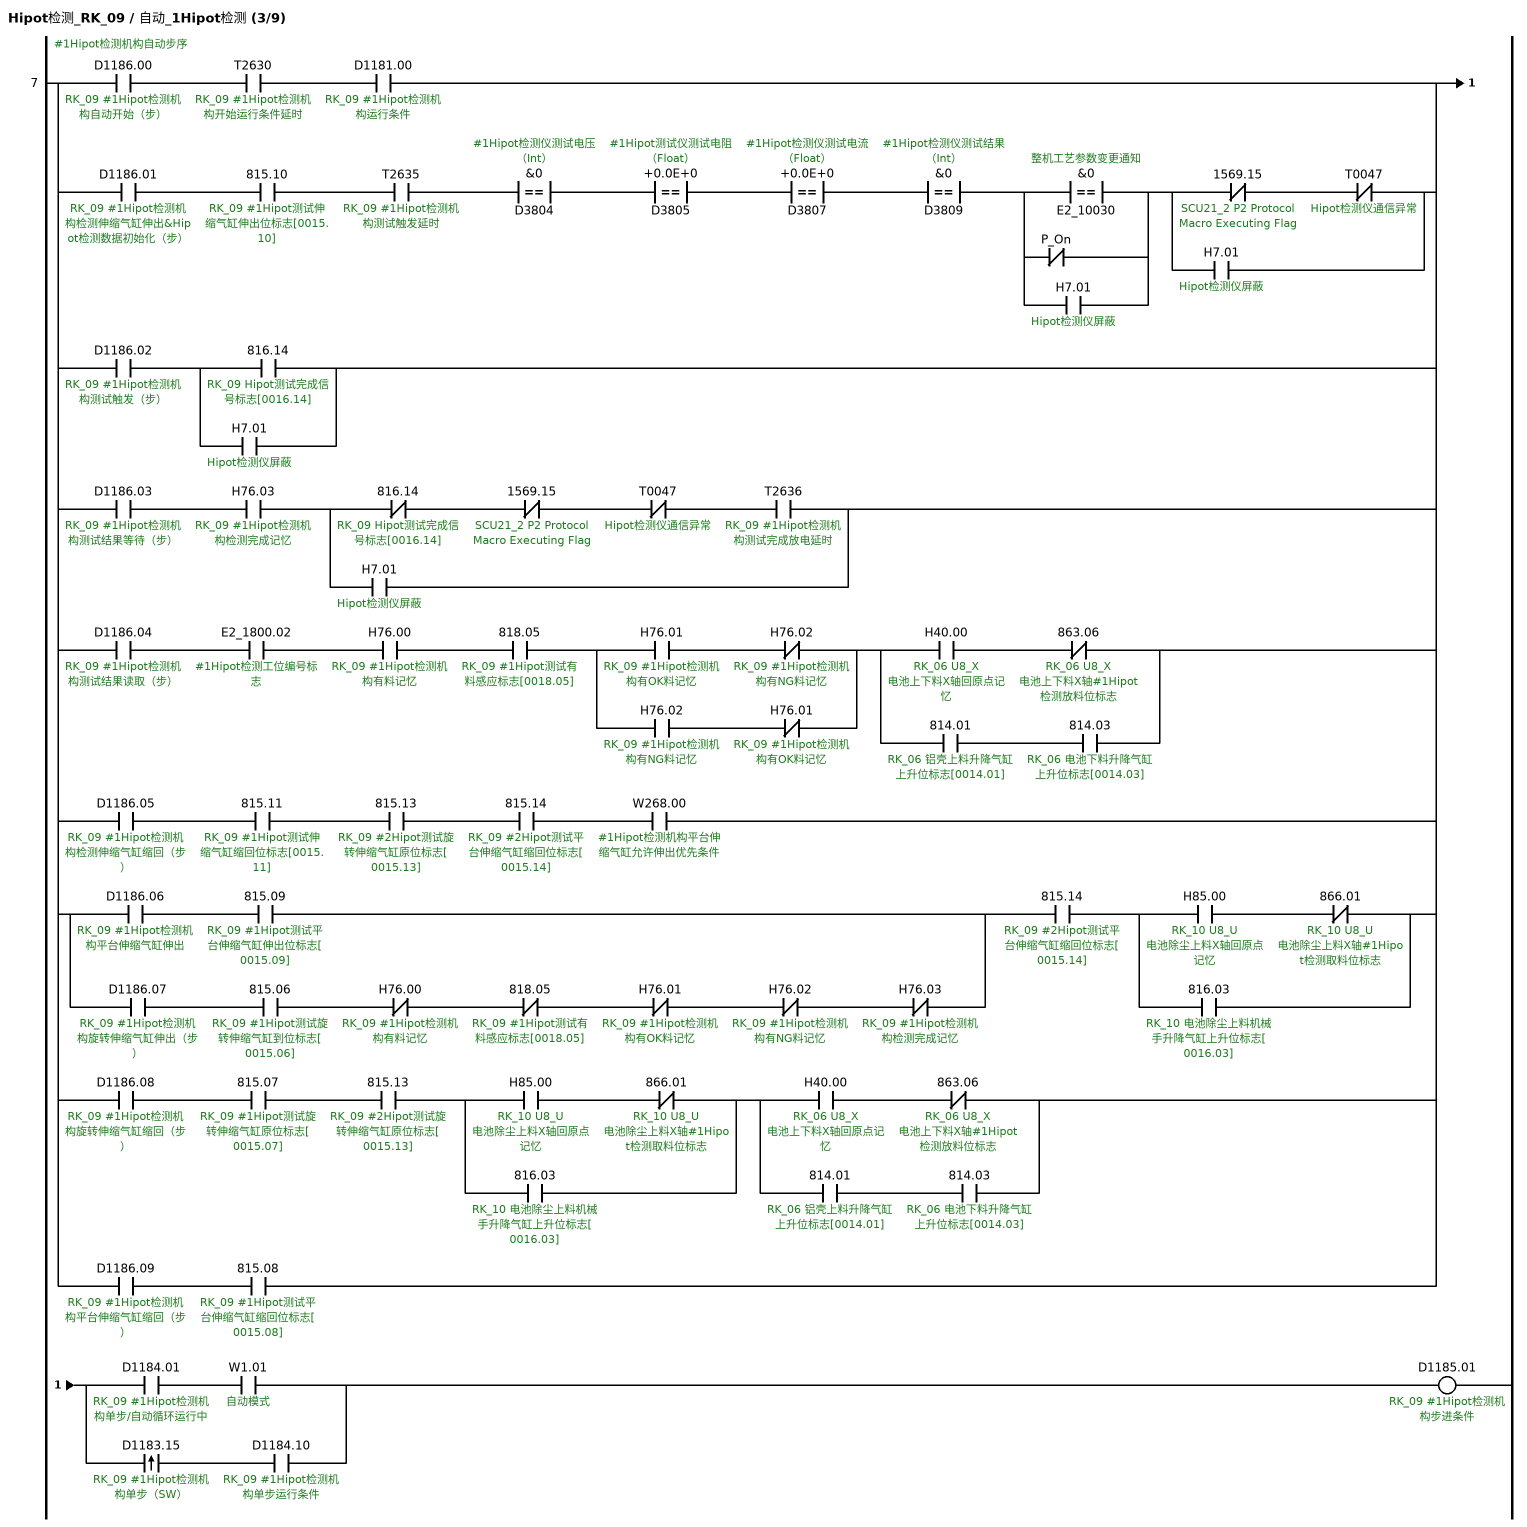
; rung 7: #1Hipot检测机构自动步序
LD D1186.00  ; RK_09 #1Hipot检测机构自动开始（步）
AND T2630  ; RK_09 #1Hipot检测机构开始运行条件延时
AND D1181.00  ; RK_09 #1Hipot检测机构运行条件
LD D1186.01  ; RK_09 #1Hipot检测机构检测伸缩气缸伸出&Hipot检测数据初始化（步）
AND 815.10  ; RK_09 #1Hipot测试伸缩气缸伸出位标志[0015.10]
AND T2635  ; RK_09 #1Hipot检测机构测试触发延时
AND=(300) &0 D3804  ; #1Hipot检测仪测试电压（Int）
AND=F(329) +0.0E+0 D3805  ; #1Hipot测试仪测试电阻（Float）
AND=F(329) +0.0E+0 D3807  ; #1Hipot检测仪测试电流（Float）
AND=(300) &0 D3809  ; #1Hipot检测仪测试结果（Int）
LD=(300) &0 E2_10030  ; 整机工艺参数变更通知
ORNOT P_On
OR H7.01  ; Hipot检测仪屏蔽
ANDLD
LDNOT 1569.15  ; SCU21_2 P2 Protocol Macro Executing Flag
ANDNOT T0047  ; Hipot检测仪通信异常
OR H7.01  ; Hipot检测仪屏蔽
ANDLD
ORLD
LD D1186.02  ; RK_09 #1Hipot检测机构测试触发（步）
LD 816.14  ; RK_09 Hipot测试完成信号标志[0016.14]
OR H7.01  ; Hipot检测仪屏蔽
ANDLD
ORLD
LD D1186.03  ; RK_09 #1Hipot检测机构测试结果等待（步）
AND H76.03  ; RK_09 #1Hipot检测机构检测完成记忆
LDNOT 816.14  ; RK_09 Hipot测试完成信号标志[0016.14]
ANDNOT 1569.15  ; SCU21_2 P2 Protocol Macro Executing Flag
ANDNOT T0047  ; Hipot检测仪通信异常
AND T2636  ; RK_09 #1Hipot检测机构测试完成放电延时
OR H7.01  ; Hipot检测仪屏蔽
ANDLD
ORLD
LD D1186.04  ; RK_09 #1Hipot检测机构测试结果读取（步）
AND E2_1800.02  ; #1Hipot检测工位编号标志
AND H76.00  ; RK_09 #1Hipot检测机构有料记忆
AND 818.05  ; RK_09 #1Hipot测试有料感应标志[0018.05]
LD H76.01  ; RK_09 #1Hipot检测机构有OK料记忆
ANDNOT H76.02  ; RK_09 #1Hipot检测机构有NG料记忆
LD H76.02  ; RK_09 #1Hipot检测机构有NG料记忆
ANDNOT H76.01  ; RK_09 #1Hipot检测机构有OK料记忆
ORLD
ANDLD
LD H40.00  ; RK_06 U8_X 电池上下料X轴回原点记忆
ANDNOT 863.06  ; RK_06 U8_X 电池上下料X轴#1Hipot检测放料位标志
LD 814.01  ; RK_06 铝壳上料升降气缸上升位标志[0014.01]
AND 814.03  ; RK_06 电池下料升降气缸上升位标志[0014.03]
ORLD
ANDLD
ORLD
LD D1186.05  ; RK_09 #1Hipot检测机构检测伸缩气缸缩回（步）
AND 815.11  ; RK_09 #1Hipot测试伸缩气缸缩回位标志[0015.11]
AND 815.13  ; RK_09 #2Hipot测试旋转伸缩气缸原位标志[0015.13]
AND 815.14  ; RK_09 #2Hipot测试平台伸缩气缸缩回位标志[0015.14]
AND W268.00  ; #1Hipot检测机构平台伸缩气缸允许伸出优先条件
ORLD
LD D1186.06  ; RK_09 #1Hipot检测机构平台伸缩气缸伸出
AND 815.09  ; RK_09 #1Hipot测试平台伸缩气缸伸出位标志[0015.09]
LD D1186.07  ; RK_09 #1Hipot检测机构旋转伸缩气缸伸出（步）
AND 815.06  ; RK_09 #1Hipot测试旋转伸缩气缸到位标志[0015.06]
ANDNOT H76.00  ; RK_09 #1Hipot检测机构有料记忆
ANDNOT 818.05  ; RK_09 #1Hipot测试有料感应标志[0018.05]
ANDNOT H76.01  ; RK_09 #1Hipot检测机构有OK料记忆
ANDNOT H76.02  ; RK_09 #1Hipot检测机构有NG料记忆
ANDNOT H76.03  ; RK_09 #1Hipot检测机构检测完成记忆
ORLD
AND 815.14  ; RK_09 #2Hipot测试平台伸缩气缸缩回位标志[0015.14]
LD H85.00  ; RK_10 U8_U 电池除尘上料X轴回原点记忆
ANDNOT 866.01  ; RK_10 U8_U 电池除尘上料X轴#1Hipot检测取料位标志
OR 816.03  ; RK_10 电池除尘上料机械手升降气缸上升位标志[0016.03]
ANDLD
ORLD
LD D1186.08  ; RK_09 #1Hipot检测机构旋转伸缩气缸缩回（步）
AND 815.07  ; RK_09 #1Hipot测试旋转伸缩气缸原位标志[0015.07]
AND 815.13  ; RK_09 #2Hipot测试旋转伸缩气缸原位标志[0015.13]
LD H85.00  ; RK_10 U8_U 电池除尘上料X轴回原点记忆
ANDNOT 866.01  ; RK_10 U8_U 电池除尘上料X轴#1Hipot检测取料位标志
OR 816.03  ; RK_10 电池除尘上料机械手升降气缸上升位标志[0016.03]
ANDLD
LD H40.00  ; RK_06 U8_X 电池上下料X轴回原点记忆
ANDNOT 863.06  ; RK_06 U8_X 电池上下料X轴#1Hipot检测放料位标志
LD 814.01  ; RK_06 铝壳上料升降气缸上升位标志[0014.01]
AND 814.03  ; RK_06 电池下料升降气缸上升位标志[0014.03]
ORLD
ANDLD
ORLD
LD D1186.09  ; RK_09 #1Hipot检测机构平台伸缩气缸缩回（步）
AND 815.08  ; RK_09 #1Hipot测试平台伸缩气缸缩回位标志[0015.08]
ORLD
LD D1184.01  ; RK_09 #1Hipot检测机构单步/自动循环运行中
AND W1.01  ; 自动模式
@LD D1183.15  ; RK_09 #1Hipot检测机构单步（SW）
AND D1184.10  ; RK_09 #1Hipot检测机构单步运行条件
ORLD
ANDLD
OUT D1185.01  ; RK_09 #1Hipot检测机构步进条件

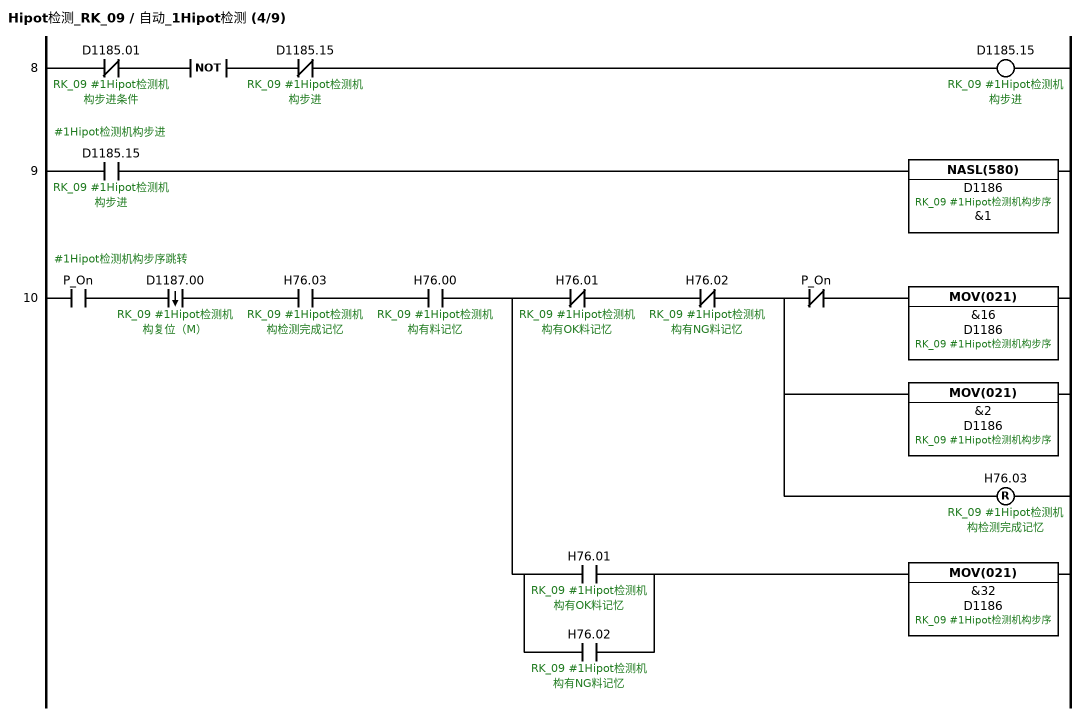
; rung 8
LDNOT D1185.01  ; RK_09 #1Hipot检测机构步进条件
NOT(520)
ANDNOT D1185.15  ; RK_09 #1Hipot检测机构步进
OUT D1185.15  ; RK_09 #1Hipot检测机构步进
; rung 9: #1Hipot检测机构步进
LD D1185.15  ; RK_09 #1Hipot检测机构步进
NASL(580) D1186 &1  ; RK_09 #1Hipot检测机构步序
; rung 10: #1Hipot检测机构步序跳转
LD P_On
%AND D1187.00  ; RK_09 #1Hipot检测机构复位（M）
AND H76.03  ; RK_09 #1Hipot检测机构检测完成记忆
AND H76.00  ; RK_09 #1Hipot检测机构有料记忆
OUT TR0
ANDNOT H76.01  ; RK_09 #1Hipot检测机构有OK料记忆
ANDNOT H76.02  ; RK_09 #1Hipot检测机构有NG料记忆
OUT TR1
ANDNOT P_On
MOV(021) &16 D1186  ; RK_09 #1Hipot检测机构步序  // RK_09 #1Hipot检测机构测试结果读取步（D1186.04）
LD TR1
MOV(021) &2 D1186  ; RK_09 #1Hipot检测机构步序  // RK_09 #1Hipot检测机构检测伸缩气缸伸出&Hipot检测数据初始化步（D1186.01）
RSET H76.03  ; RK_09 #1Hipot检测机构检测完成记忆
LD TR0
LD H76.01  ; RK_09 #1Hipot检测机构有OK料记忆
OR H76.02  ; RK_09 #1Hipot检测机构有NG料记忆
ANDLD
MOV(021) &32 D1186  ; RK_09 #1Hipot检测机构步序  // RK_09 #1Hipot检测机构检测伸缩气缸缩回步（D1186.05）

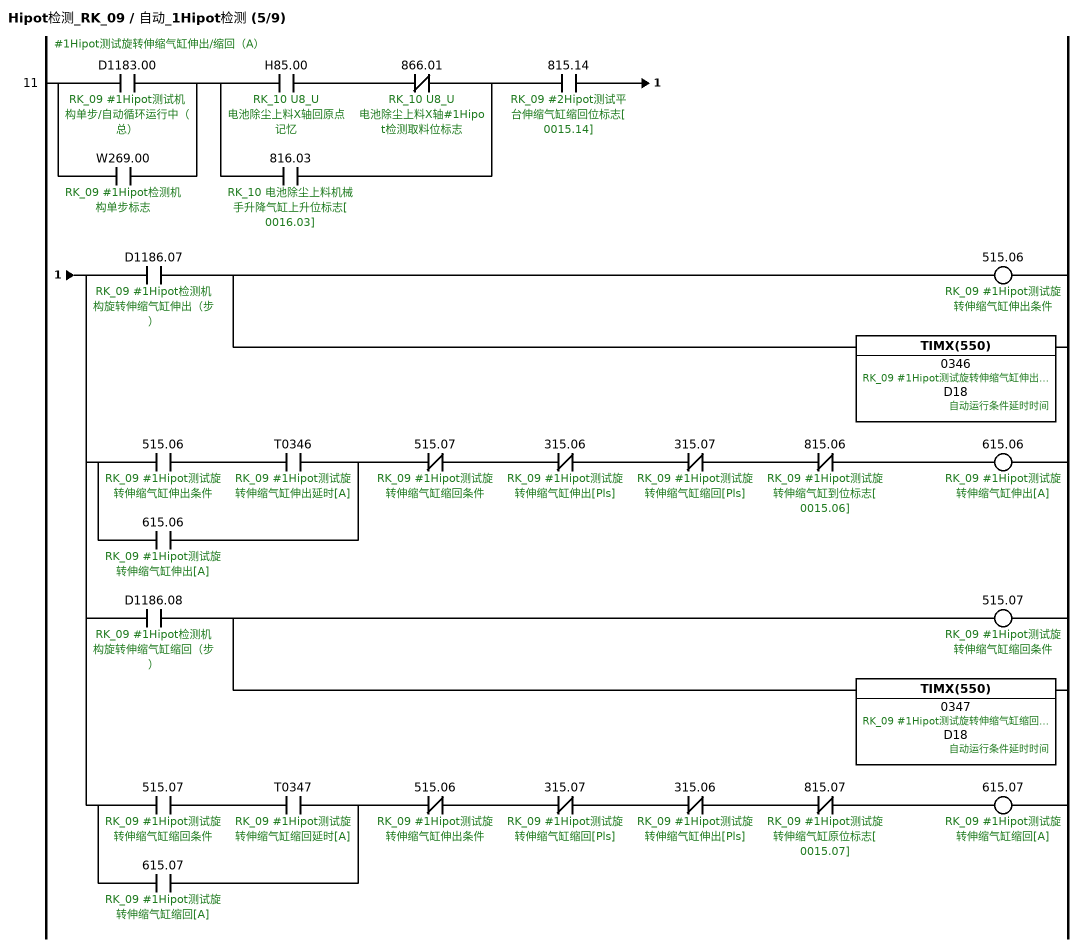
; rung 11: #1Hipot测试旋转伸缩气缸伸出/缩回（A）
LD D1183.00  ; RK_09 #1Hipot测试机构单步/自动循环运行中（总）
OR W269.00  ; RK_09 #1Hipot检测机构单步标志
LD H85.00  ; RK_10 U8_U 电池除尘上料X轴回原点记忆
ANDNOT 866.01  ; RK_10 U8_U 电池除尘上料X轴#1Hipot检测取料位标志
OR 816.03  ; RK_10 电池除尘上料机械手升降气缸上升位标志[0016.03]
ANDLD
AND 815.14  ; RK_09 #2Hipot测试平台伸缩气缸缩回位标志[0015.14]
OUT TR0
AND D1186.07  ; RK_09 #1Hipot检测机构旋转伸缩气缸伸出（步）
OUT 515.06  ; RK_09 #1Hipot测试旋转伸缩气缸伸出条件
TIMX(550) 0346 D18  ; 自动运行条件延时时间, RK_09 #1Hipot测试旋转伸缩气缸伸出延时[A]
LD TR0
LD 515.06  ; RK_09 #1Hipot测试旋转伸缩气缸伸出条件
AND T0346  ; RK_09 #1Hipot测试旋转伸缩气缸伸出延时[A]
OR 615.06  ; RK_09 #1Hipot测试旋转伸缩气缸伸出[A]
ANDLD
ANDNOT 515.07  ; RK_09 #1Hipot测试旋转伸缩气缸缩回条件
ANDNOT 315.06  ; RK_09 #1Hipot测试旋转伸缩气缸伸出[Pls]
ANDNOT 315.07  ; RK_09 #1Hipot测试旋转伸缩气缸缩回[Pls]
ANDNOT 815.06  ; RK_09 #1Hipot测试旋转伸缩气缸到位标志[0015.06]
OUT 615.06  ; RK_09 #1Hipot测试旋转伸缩气缸伸出[A]
LD TR0
AND D1186.08  ; RK_09 #1Hipot检测机构旋转伸缩气缸缩回（步）
OUT 515.07  ; RK_09 #1Hipot测试旋转伸缩气缸缩回条件
TIMX(550) 0347 D18  ; 自动运行条件延时时间, RK_09 #1Hipot测试旋转伸缩气缸缩回延时[A]
LD TR0
LD 515.07  ; RK_09 #1Hipot测试旋转伸缩气缸缩回条件
AND T0347  ; RK_09 #1Hipot测试旋转伸缩气缸缩回延时[A]
OR 615.07  ; RK_09 #1Hipot测试旋转伸缩气缸缩回[A]
ANDLD
ANDNOT 515.06  ; RK_09 #1Hipot测试旋转伸缩气缸伸出条件
ANDNOT 315.07  ; RK_09 #1Hipot测试旋转伸缩气缸缩回[Pls]
ANDNOT 315.06  ; RK_09 #1Hipot测试旋转伸缩气缸伸出[Pls]
ANDNOT 815.07  ; RK_09 #1Hipot测试旋转伸缩气缸原位标志[0015.07]
OUT 615.07  ; RK_09 #1Hipot测试旋转伸缩气缸缩回[A]

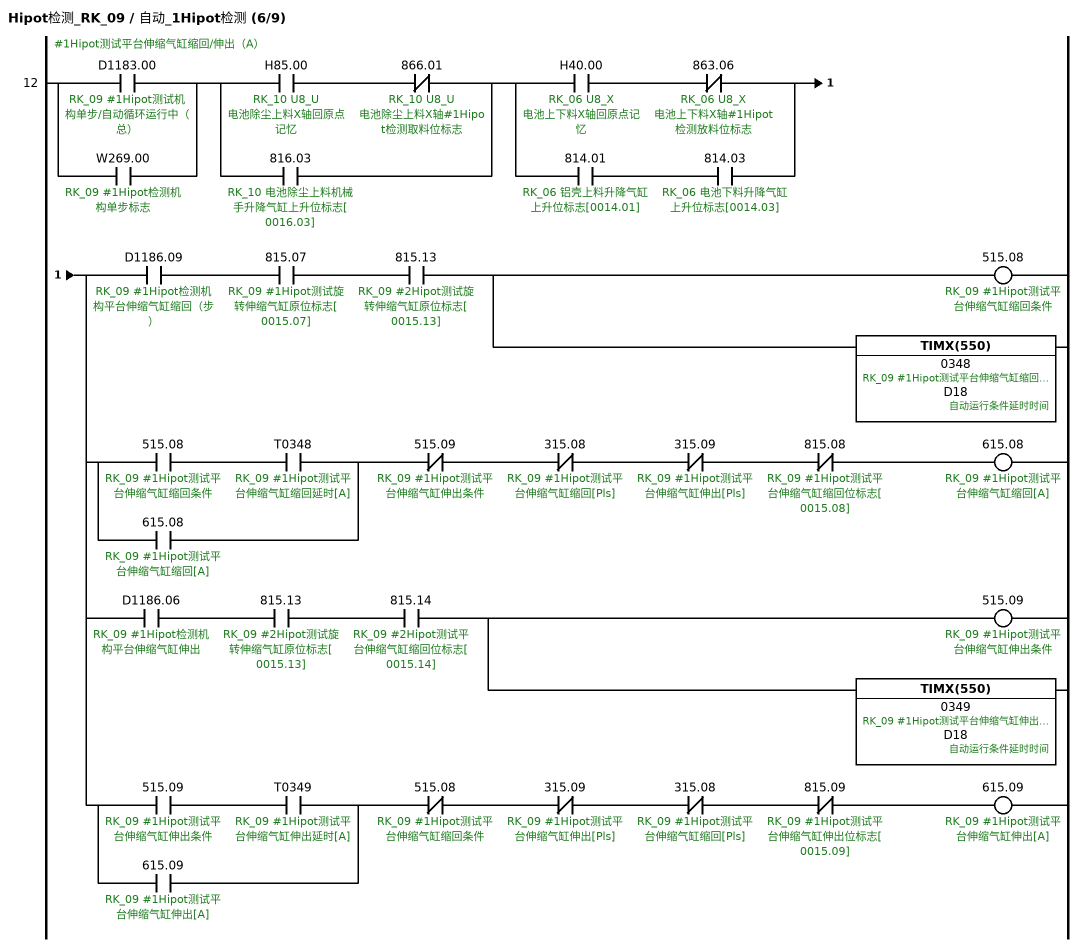
; rung 12: #1Hipot测试平台伸缩气缸缩回/伸出（A）
LD D1183.00  ; RK_09 #1Hipot测试机构单步/自动循环运行中（总）
OR W269.00  ; RK_09 #1Hipot检测机构单步标志
LD H85.00  ; RK_10 U8_U 电池除尘上料X轴回原点记忆
ANDNOT 866.01  ; RK_10 U8_U 电池除尘上料X轴#1Hipot检测取料位标志
OR 816.03  ; RK_10 电池除尘上料机械手升降气缸上升位标志[0016.03]
ANDLD
LD H40.00  ; RK_06 U8_X 电池上下料X轴回原点记忆
ANDNOT 863.06  ; RK_06 U8_X 电池上下料X轴#1Hipot检测放料位标志
LD 814.01  ; RK_06 铝壳上料升降气缸上升位标志[0014.01]
AND 814.03  ; RK_06 电池下料升降气缸上升位标志[0014.03]
ORLD
ANDLD
OUT TR0
AND D1186.09  ; RK_09 #1Hipot检测机构平台伸缩气缸缩回（步）
AND 815.07  ; RK_09 #1Hipot测试旋转伸缩气缸原位标志[0015.07]
AND 815.13  ; RK_09 #2Hipot测试旋转伸缩气缸原位标志[0015.13]
OUT 515.08  ; RK_09 #1Hipot测试平台伸缩气缸缩回条件
TIMX(550) 0348 D18  ; 自动运行条件延时时间, RK_09 #1Hipot测试平台伸缩气缸缩回延时[A]
LD TR0
LD 515.08  ; RK_09 #1Hipot测试平台伸缩气缸缩回条件
AND T0348  ; RK_09 #1Hipot测试平台伸缩气缸缩回延时[A]
OR 615.08  ; RK_09 #1Hipot测试平台伸缩气缸缩回[A]
ANDLD
ANDNOT 515.09  ; RK_09 #1Hipot测试平台伸缩气缸伸出条件
ANDNOT 315.08  ; RK_09 #1Hipot测试平台伸缩气缸缩回[Pls]
ANDNOT 315.09  ; RK_09 #1Hipot测试平台伸缩气缸伸出[Pls]
ANDNOT 815.08  ; RK_09 #1Hipot测试平台伸缩气缸缩回位标志[0015.08]
OUT 615.08  ; RK_09 #1Hipot测试平台伸缩气缸缩回[A]
LD TR0
AND D1186.06  ; RK_09 #1Hipot检测机构平台伸缩气缸伸出
AND 815.13  ; RK_09 #2Hipot测试旋转伸缩气缸原位标志[0015.13]
AND 815.14  ; RK_09 #2Hipot测试平台伸缩气缸缩回位标志[0015.14]
OUT 515.09  ; RK_09 #1Hipot测试平台伸缩气缸伸出条件
TIMX(550) 0349 D18  ; 自动运行条件延时时间, RK_09 #1Hipot测试平台伸缩气缸伸出延时[A]
LD TR0
LD 515.09  ; RK_09 #1Hipot测试平台伸缩气缸伸出条件
AND T0349  ; RK_09 #1Hipot测试平台伸缩气缸伸出延时[A]
OR 615.09  ; RK_09 #1Hipot测试平台伸缩气缸伸出[A]
ANDLD
ANDNOT 515.08  ; RK_09 #1Hipot测试平台伸缩气缸缩回条件
ANDNOT 315.09  ; RK_09 #1Hipot测试平台伸缩气缸伸出[Pls]
ANDNOT 315.08  ; RK_09 #1Hipot测试平台伸缩气缸缩回[Pls]
ANDNOT 815.09  ; RK_09 #1Hipot测试平台伸缩气缸伸出位标志[0015.09]
OUT 615.09  ; RK_09 #1Hipot测试平台伸缩气缸伸出[A]

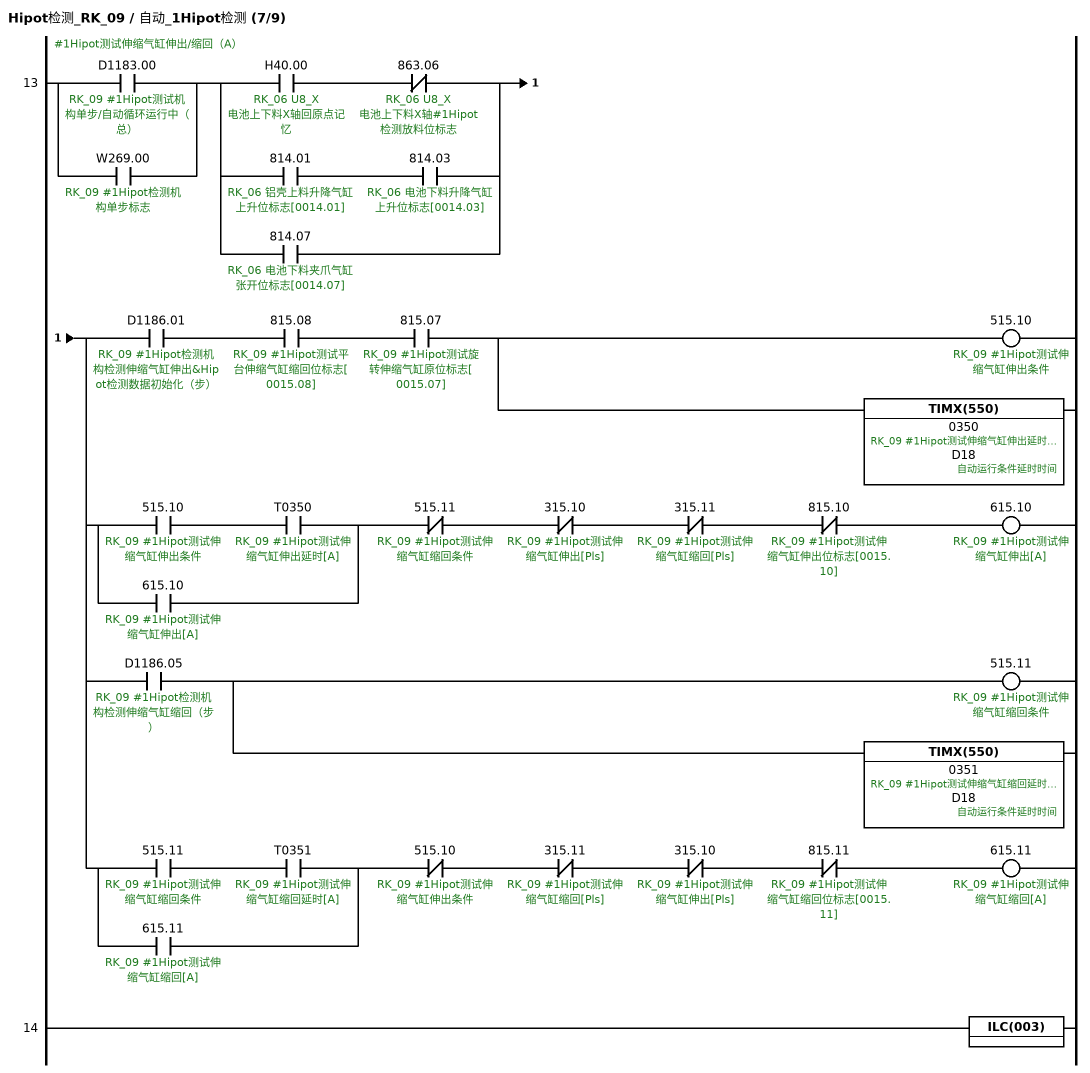
; rung 13: #1Hipot测试伸缩气缸伸出/缩回（A）
LD D1183.00  ; RK_09 #1Hipot测试机构单步/自动循环运行中（总）
OR W269.00  ; RK_09 #1Hipot检测机构单步标志
LD H40.00  ; RK_06 U8_X 电池上下料X轴回原点记忆
ANDNOT 863.06  ; RK_06 U8_X 电池上下料X轴#1Hipot检测放料位标志
LD 814.01  ; RK_06 铝壳上料升降气缸上升位标志[0014.01]
AND 814.03  ; RK_06 电池下料升降气缸上升位标志[0014.03]
ORLD
OR 814.07  ; RK_06 电池下料夹爪气缸张开位标志[0014.07]
ANDLD
OUT TR0
AND D1186.01  ; RK_09 #1Hipot检测机构检测伸缩气缸伸出&Hipot检测数据初始化（步）
AND 815.08  ; RK_09 #1Hipot测试平台伸缩气缸缩回位标志[0015.08]
AND 815.07  ; RK_09 #1Hipot测试旋转伸缩气缸原位标志[0015.07]
OUT 515.10  ; RK_09 #1Hipot测试伸缩气缸伸出条件
TIMX(550) 0350 D18  ; 自动运行条件延时时间, RK_09 #1Hipot测试伸缩气缸伸出延时[A]
LD TR0
LD 515.10  ; RK_09 #1Hipot测试伸缩气缸伸出条件
AND T0350  ; RK_09 #1Hipot测试伸缩气缸伸出延时[A]
OR 615.10  ; RK_09 #1Hipot测试伸缩气缸伸出[A]
ANDLD
ANDNOT 515.11  ; RK_09 #1Hipot测试伸缩气缸缩回条件
ANDNOT 315.10  ; RK_09 #1Hipot测试伸缩气缸伸出[Pls]
ANDNOT 315.11  ; RK_09 #1Hipot测试伸缩气缸缩回[Pls]
ANDNOT 815.10  ; RK_09 #1Hipot测试伸缩气缸伸出位标志[0015.10]
OUT 615.10  ; RK_09 #1Hipot测试伸缩气缸伸出[A]
LD TR0
AND D1186.05  ; RK_09 #1Hipot检测机构检测伸缩气缸缩回（步）
OUT 515.11  ; RK_09 #1Hipot测试伸缩气缸缩回条件
TIMX(550) 0351 D18  ; 自动运行条件延时时间, RK_09 #1Hipot测试伸缩气缸缩回延时[A]
LD TR0
LD 515.11  ; RK_09 #1Hipot测试伸缩气缸缩回条件
AND T0351  ; RK_09 #1Hipot测试伸缩气缸缩回延时[A]
OR 615.11  ; RK_09 #1Hipot测试伸缩气缸缩回[A]
ANDLD
ANDNOT 515.10  ; RK_09 #1Hipot测试伸缩气缸伸出条件
ANDNOT 315.11  ; RK_09 #1Hipot测试伸缩气缸缩回[Pls]
ANDNOT 315.10  ; RK_09 #1Hipot测试伸缩气缸伸出[Pls]
ANDNOT 815.11  ; RK_09 #1Hipot测试伸缩气缸缩回位标志[0015.11]
OUT 615.11  ; RK_09 #1Hipot测试伸缩气缸缩回[A]
; rung 14
ILC(003)

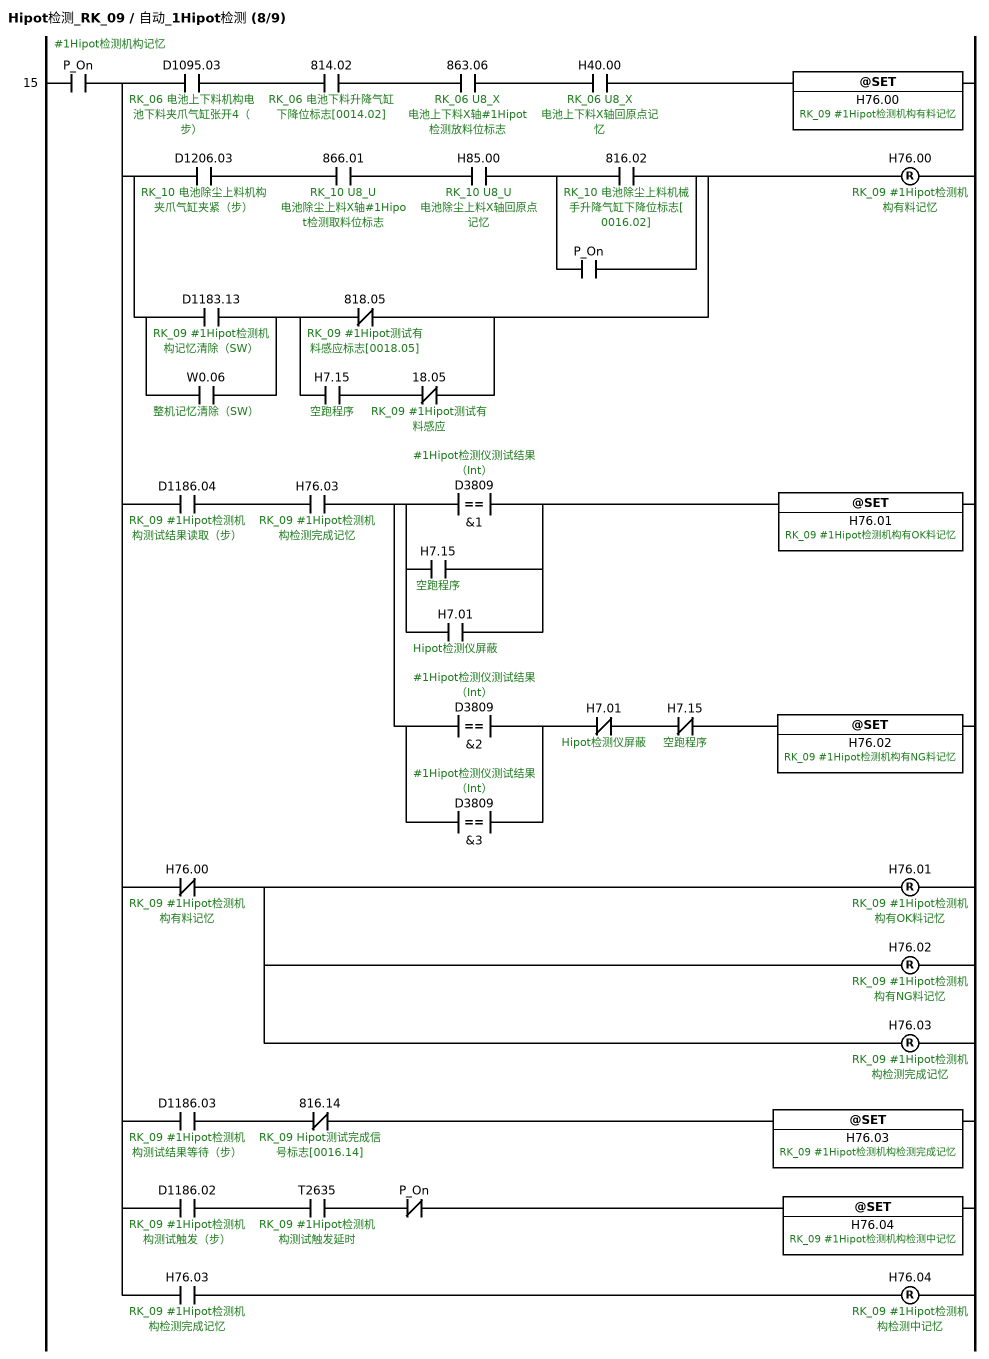
; rung 15: #1Hipot检测机构记忆
LD P_On
OUT TR0
AND D1095.03  ; RK_06 电池上下料机构电池下料夹爪气缸张开4（步）
AND 814.02  ; RK_06 电池下料升降气缸下降位标志[0014.02]
AND 863.06  ; RK_06 U8_X 电池上下料X轴#1Hipot检测放料位标志
AND H40.00  ; RK_06 U8_X 电池上下料X轴回原点记忆
@SET H76.00  ; RK_09 #1Hipot检测机构有料记忆
LD TR0
LD D1206.03  ; RK_10 电池除尘上料机构夹爪气缸夹紧（步）
AND 866.01  ; RK_10 U8_U 电池除尘上料X轴#1Hipot检测取料位标志
AND H85.00  ; RK_10 U8_U 电池除尘上料X轴回原点记忆
LD 816.02  ; RK_10 电池除尘上料机械手升降气缸下降位标志[0016.02]
OR P_On
ANDLD
LD D1183.13  ; RK_09 #1Hipot检测机构记忆清除（SW）
OR W0.06  ; 整机记忆清除（SW）
LDNOT 818.05  ; RK_09 #1Hipot测试有料感应标志[0018.05]
LD H7.15  ; 空跑程序
ANDNOT 18.05  ; RK_09 #1Hipot测试有料感应
ORLD
ANDLD
ORLD
ANDLD
RSET H76.00  ; RK_09 #1Hipot检测机构有料记忆
LD TR0
AND D1186.04  ; RK_09 #1Hipot检测机构测试结果读取（步）
AND H76.03  ; RK_09 #1Hipot检测机构检测完成记忆
OUT TR1
LD=(300) D3809 &1  ; #1Hipot检测仪测试结果（Int）
OR H7.15  ; 空跑程序
OR H7.01  ; Hipot检测仪屏蔽
ANDLD
@SET H76.01  ; RK_09 #1Hipot检测机构有OK料记忆
LD TR1
LD=(300) D3809 &2  ; #1Hipot检测仪测试结果（Int）
OR=(300) D3809 &3  ; #1Hipot检测仪测试结果（Int）
ANDLD
ANDNOT H7.01  ; Hipot检测仪屏蔽
ANDNOT H7.15  ; 空跑程序
@SET H76.02  ; RK_09 #1Hipot检测机构有NG料记忆
LD TR0
ANDNOT H76.00  ; RK_09 #1Hipot检测机构有料记忆
RSET H76.01  ; RK_09 #1Hipot检测机构有OK料记忆
RSET H76.02  ; RK_09 #1Hipot检测机构有NG料记忆
RSET H76.03  ; RK_09 #1Hipot检测机构检测完成记忆
LD TR0
AND D1186.03  ; RK_09 #1Hipot检测机构测试结果等待（步）
ANDNOT 816.14  ; RK_09 Hipot测试完成信号标志[0016.14]
@SET H76.03  ; RK_09 #1Hipot检测机构检测完成记忆
LD TR0
AND D1186.02  ; RK_09 #1Hipot检测机构测试触发（步）
AND T2635  ; RK_09 #1Hipot检测机构测试触发延时
ANDNOT P_On
@SET H76.04  ; RK_09 #1Hipot检测机构检测中记忆
LD TR0
AND H76.03  ; RK_09 #1Hipot检测机构检测完成记忆
RSET H76.04  ; RK_09 #1Hipot检测机构检测中记忆

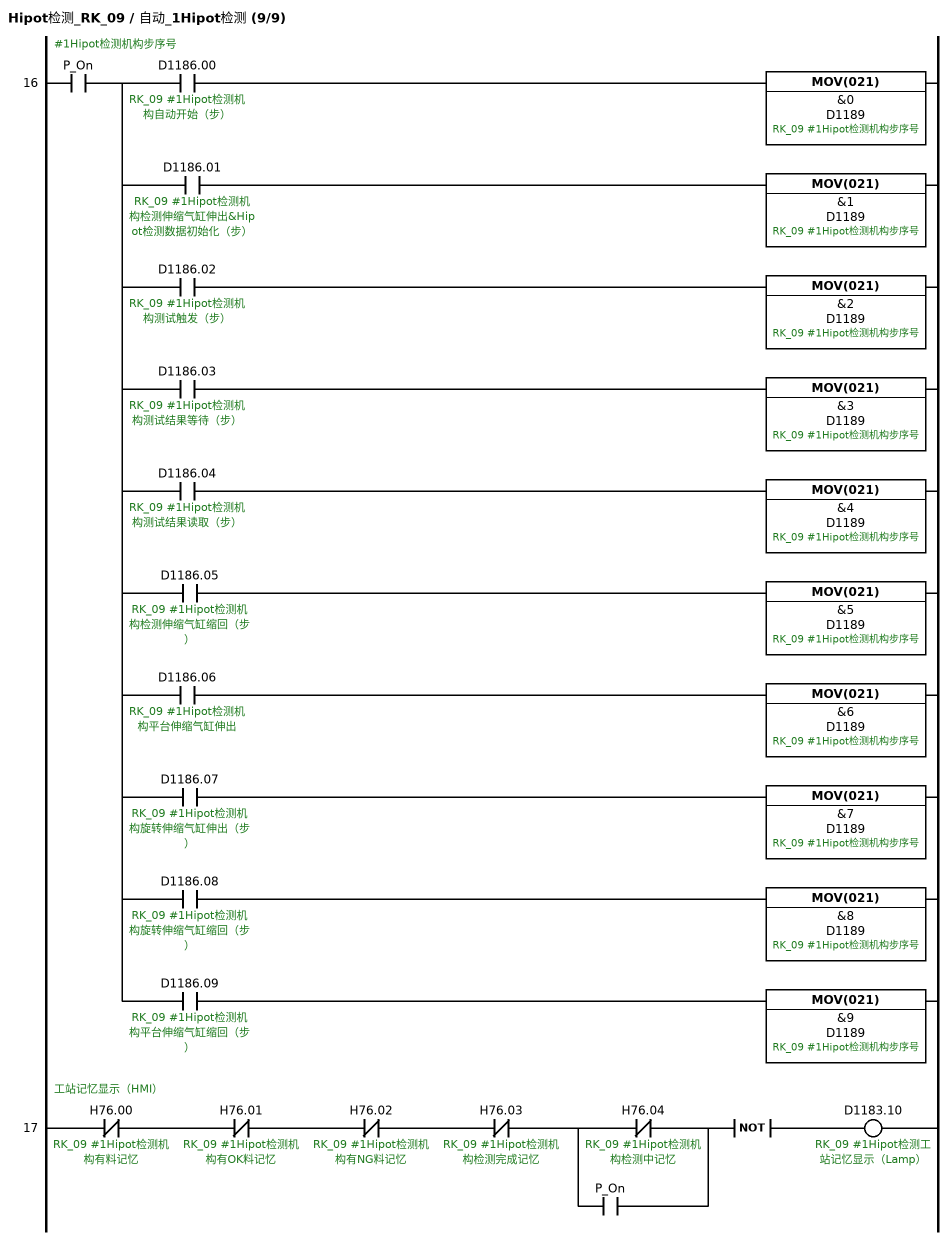
; rung 16: #1Hipot检测机构步序号
LD P_On
OUT TR0
AND D1186.00  ; RK_09 #1Hipot检测机构自动开始（步）
MOV(021) &0 D1189  ; RK_09 #1Hipot检测机构步序号
LD TR0
AND D1186.01  ; RK_09 #1Hipot检测机构检测伸缩气缸伸出&Hipot检测数据初始化（步）
MOV(021) &1 D1189  ; RK_09 #1Hipot检测机构步序号
LD TR0
AND D1186.02  ; RK_09 #1Hipot检测机构测试触发（步）
MOV(021) &2 D1189  ; RK_09 #1Hipot检测机构步序号
LD TR0
AND D1186.03  ; RK_09 #1Hipot检测机构测试结果等待（步）
MOV(021) &3 D1189  ; RK_09 #1Hipot检测机构步序号
LD TR0
AND D1186.04  ; RK_09 #1Hipot检测机构测试结果读取（步）
MOV(021) &4 D1189  ; RK_09 #1Hipot检测机构步序号
LD TR0
AND D1186.05  ; RK_09 #1Hipot检测机构检测伸缩气缸缩回（步）
MOV(021) &5 D1189  ; RK_09 #1Hipot检测机构步序号
LD TR0
AND D1186.06  ; RK_09 #1Hipot检测机构平台伸缩气缸伸出
MOV(021) &6 D1189  ; RK_09 #1Hipot检测机构步序号
LD TR0
AND D1186.07  ; RK_09 #1Hipot检测机构旋转伸缩气缸伸出（步）
MOV(021) &7 D1189  ; RK_09 #1Hipot检测机构步序号
LD TR0
AND D1186.08  ; RK_09 #1Hipot检测机构旋转伸缩气缸缩回（步）
MOV(021) &8 D1189  ; RK_09 #1Hipot检测机构步序号
LD TR0
AND D1186.09  ; RK_09 #1Hipot检测机构平台伸缩气缸缩回（步）
MOV(021) &9 D1189  ; RK_09 #1Hipot检测机构步序号
; rung 17: 工站记忆显示（HMI）
LDNOT H76.00  ; RK_09 #1Hipot检测机构有料记忆
ANDNOT H76.01  ; RK_09 #1Hipot检测机构有OK料记忆
ANDNOT H76.02  ; RK_09 #1Hipot检测机构有NG料记忆
ANDNOT H76.03  ; RK_09 #1Hipot检测机构检测完成记忆
LDNOT H76.04  ; RK_09 #1Hipot检测机构检测中记忆
OR P_On
ANDLD
NOT(520)
OUT D1183.10  ; RK_09 #1Hipot检测工站记忆显示（Lamp）

### Section 自动_2Hipot检测

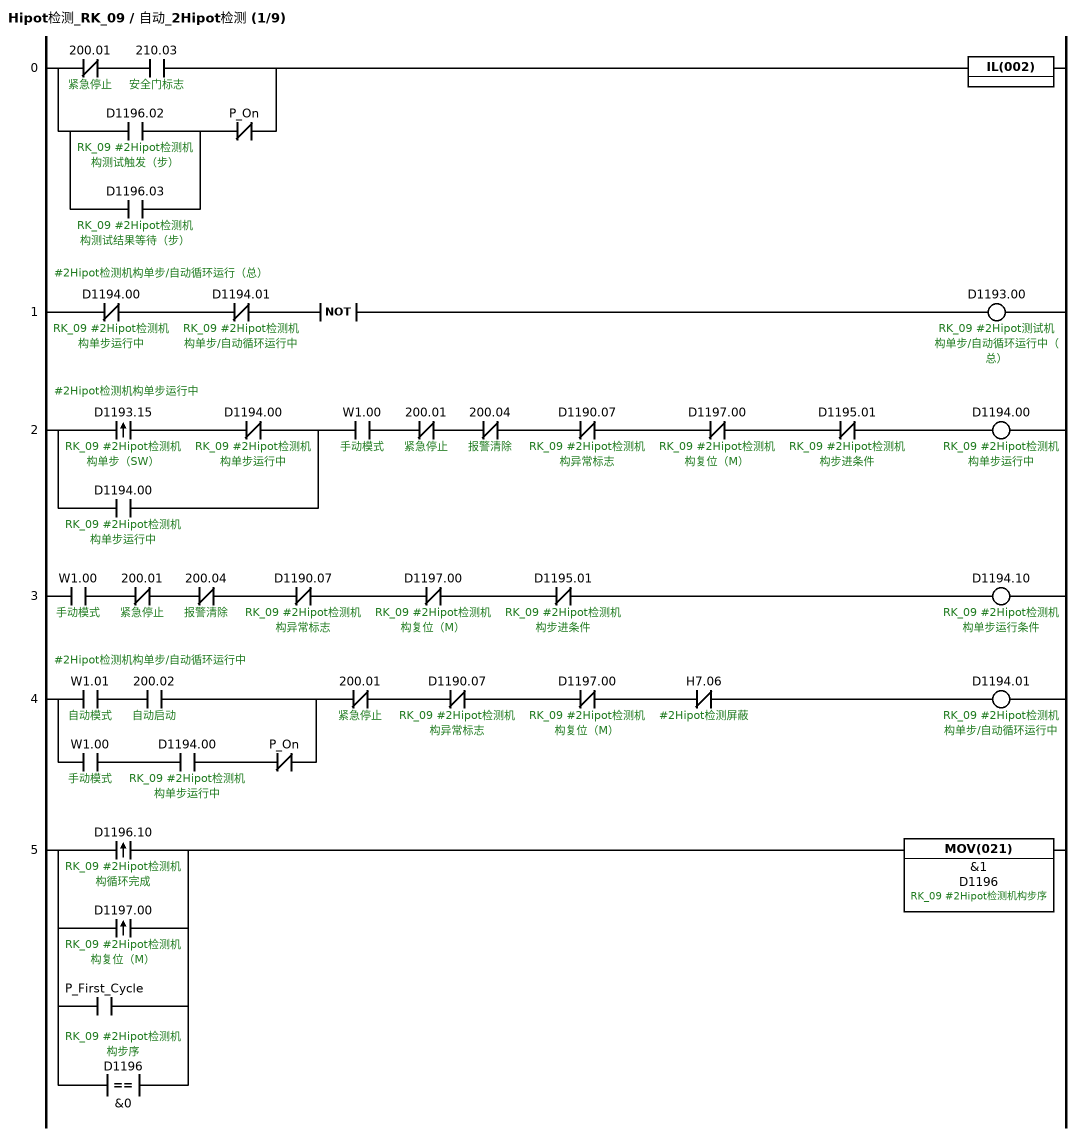
; rung 0
LDNOT 200.01  ; 紧急停止
AND 210.03  ; 安全门标志
LD D1196.02  ; RK_09 #2Hipot检测机构测试触发（步）
OR D1196.03  ; RK_09 #2Hipot检测机构测试结果等待（步）
ANDNOT P_On  // Hipot测试触发后，急停|安全门打开情况下测试继续，直到有测试完成信号！
ORLD
IL(002)
; rung 1: #2Hipot检测机构单步/自动循环运行（总）
LDNOT D1194.00  ; RK_09 #2Hipot检测机构单步运行中
ANDNOT D1194.01  ; RK_09 #2Hipot检测机构单步/自动循环运行中
NOT(520)
OUT D1193.00  ; RK_09 #2Hipot测试机构单步/自动循环运行中（总）
; rung 2: #2Hipot检测机构单步运行中
@LD D1193.15  ; RK_09 #2Hipot检测机构单步（SW）
ANDNOT D1194.00  ; RK_09 #2Hipot检测机构单步运行中
OR D1194.00  ; RK_09 #2Hipot检测机构单步运行中
AND W1.00  ; 手动模式
ANDNOT 200.01  ; 紧急停止
ANDNOT 200.04  ; 报警清除
ANDNOT D1190.07  ; RK_09 #2Hipot检测机构异常标志
ANDNOT D1197.00  ; RK_09 #2Hipot检测机构复位（M）
ANDNOT D1195.01  ; RK_09 #2Hipot检测机构步进条件
OUT D1194.00  ; RK_09 #2Hipot检测机构单步运行中
; rung 3
LD W1.00  ; 手动模式
ANDNOT 200.01  ; 紧急停止
ANDNOT 200.04  ; 报警清除
ANDNOT D1190.07  ; RK_09 #2Hipot检测机构异常标志
ANDNOT D1197.00  ; RK_09 #2Hipot检测机构复位（M）
ANDNOT D1195.01  ; RK_09 #2Hipot检测机构步进条件
OUT D1194.10  ; RK_09 #2Hipot检测机构单步运行条件
; rung 4: #2Hipot检测机构单步/自动循环运行中
LD W1.01  ; 自动模式
AND 200.02  ; 自动启动
LD W1.00  ; 手动模式
AND D1194.00  ; RK_09 #2Hipot检测机构单步运行中
ANDNOT P_On
ORLD
ANDNOT 200.01  ; 紧急停止
ANDNOT D1190.07  ; RK_09 #2Hipot检测机构异常标志
ANDNOT D1197.00  ; RK_09 #2Hipot检测机构复位（M）
ANDNOT H7.06  ; #2Hipot检测屏蔽
OUT D1194.01  ; RK_09 #2Hipot检测机构单步/自动循环运行中
; rung 5
@LD D1196.10  ; RK_09 #2Hipot检测机构循环完成
@OR D1197.00  ; RK_09 #2Hipot检测机构复位（M）
OR P_First_Cycle
OR=(300) D1196 &0  ; RK_09 #2Hipot检测机构步序
MOV(021) &1 D1196  ; RK_09 #2Hipot检测机构步序

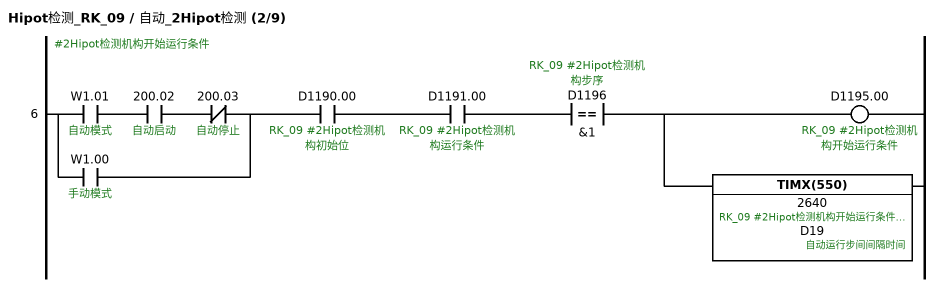
; rung 6: #2Hipot检测机构开始运行条件
LD W1.01  ; 自动模式
AND 200.02  ; 自动启动
ANDNOT 200.03  ; 自动停止
OR W1.00  ; 手动模式
AND D1190.00  ; RK_09 #2Hipot检测机构初始位
AND D1191.00  ; RK_09 #2Hipot检测机构运行条件
AND=(300) D1196 &1  ; RK_09 #2Hipot检测机构步序
OUT D1195.00  ; RK_09 #2Hipot检测机构开始运行条件
TIMX(550) 2640 D19  ; 自动运行步间间隔时间, RK_09 #2Hipot检测机构开始运行条件延时

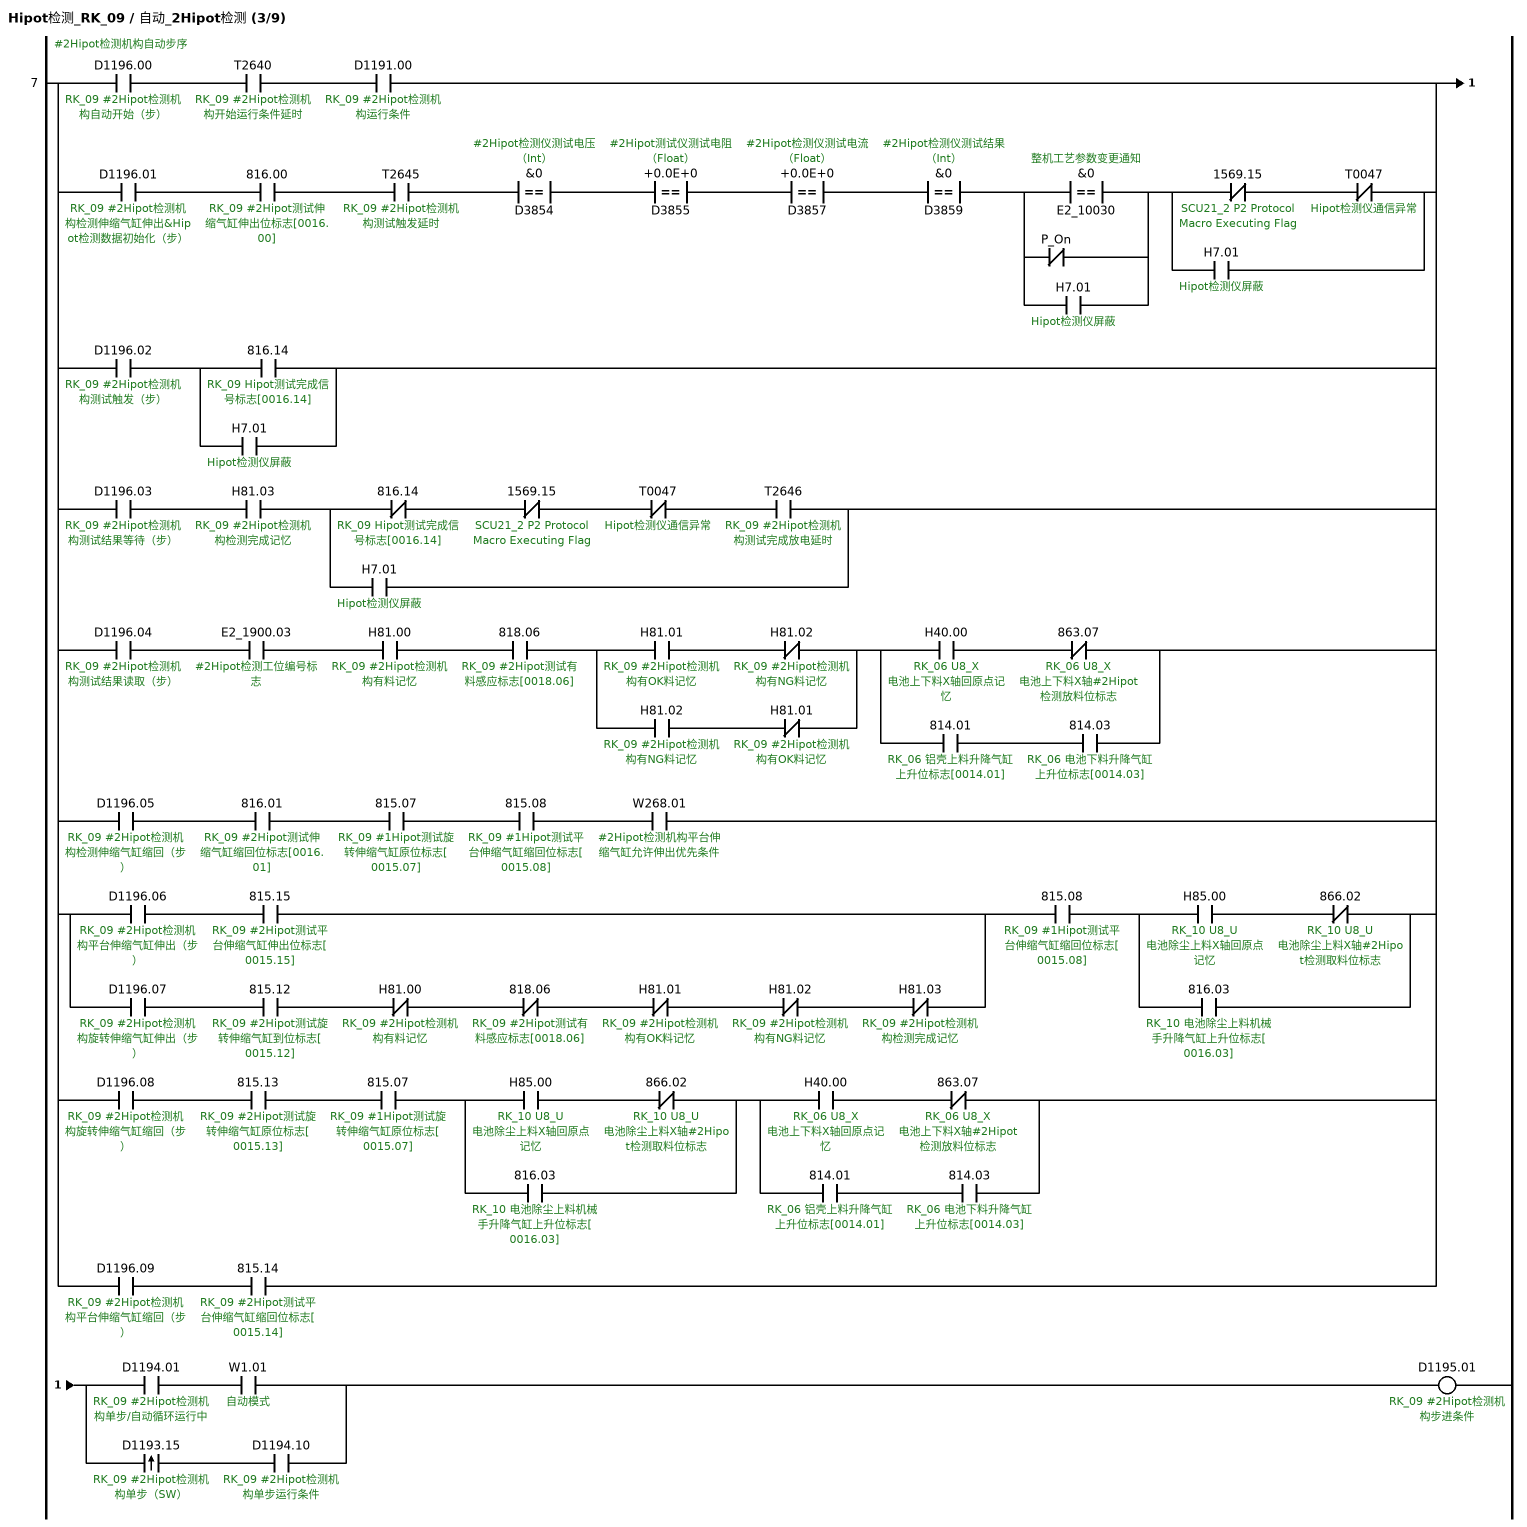
; rung 7: #2Hipot检测机构自动步序
LD D1196.00  ; RK_09 #2Hipot检测机构自动开始（步）
AND T2640  ; RK_09 #2Hipot检测机构开始运行条件延时
AND D1191.00  ; RK_09 #2Hipot检测机构运行条件
LD D1196.01  ; RK_09 #2Hipot检测机构检测伸缩气缸伸出&Hipot检测数据初始化（步）
AND 816.00  ; RK_09 #2Hipot测试伸缩气缸伸出位标志[0016.00]
AND T2645  ; RK_09 #2Hipot检测机构测试触发延时
AND=(300) &0 D3854  ; #2Hipot检测仪测试电压（Int）
AND=F(329) +0.0E+0 D3855  ; #2Hipot测试仪测试电阻（Float）
AND=F(329) +0.0E+0 D3857  ; #2Hipot检测仪测试电流（Float）
AND=(300) &0 D3859  ; #2Hipot检测仪测试结果（Int）
LD=(300) &0 E2_10030  ; 整机工艺参数变更通知
ORNOT P_On
OR H7.01  ; Hipot检测仪屏蔽
ANDLD
LDNOT 1569.15  ; SCU21_2 P2 Protocol Macro Executing Flag
ANDNOT T0047  ; Hipot检测仪通信异常
OR H7.01  ; Hipot检测仪屏蔽
ANDLD
ORLD
LD D1196.02  ; RK_09 #2Hipot检测机构测试触发（步）
LD 816.14  ; RK_09 Hipot测试完成信号标志[0016.14]
OR H7.01  ; Hipot检测仪屏蔽
ANDLD
ORLD
LD D1196.03  ; RK_09 #2Hipot检测机构测试结果等待（步）
AND H81.03  ; RK_09 #2Hipot检测机构检测完成记忆
LDNOT 816.14  ; RK_09 Hipot测试完成信号标志[0016.14]
ANDNOT 1569.15  ; SCU21_2 P2 Protocol Macro Executing Flag
ANDNOT T0047  ; Hipot检测仪通信异常
AND T2646  ; RK_09 #2Hipot检测机构测试完成放电延时
OR H7.01  ; Hipot检测仪屏蔽
ANDLD
ORLD
LD D1196.04  ; RK_09 #2Hipot检测机构测试结果读取（步）
AND E2_1900.03  ; #2Hipot检测工位编号标志
AND H81.00  ; RK_09 #2Hipot检测机构有料记忆
AND 818.06  ; RK_09 #2Hipot测试有料感应标志[0018.06]
LD H81.01  ; RK_09 #2Hipot检测机构有OK料记忆
ANDNOT H81.02  ; RK_09 #2Hipot检测机构有NG料记忆
LD H81.02  ; RK_09 #2Hipot检测机构有NG料记忆
ANDNOT H81.01  ; RK_09 #2Hipot检测机构有OK料记忆
ORLD
ANDLD
LD H40.00  ; RK_06 U8_X 电池上下料X轴回原点记忆
ANDNOT 863.07  ; RK_06 U8_X 电池上下料X轴#2Hipot检测放料位标志
LD 814.01  ; RK_06 铝壳上料升降气缸上升位标志[0014.01]
AND 814.03  ; RK_06 电池下料升降气缸上升位标志[0014.03]
ORLD
ANDLD
ORLD
LD D1196.05  ; RK_09 #2Hipot检测机构检测伸缩气缸缩回（步）
AND 816.01  ; RK_09 #2Hipot测试伸缩气缸缩回位标志[0016.01]
AND 815.07  ; RK_09 #1Hipot测试旋转伸缩气缸原位标志[0015.07]
AND 815.08  ; RK_09 #1Hipot测试平台伸缩气缸缩回位标志[0015.08]
AND W268.01  ; #2Hipot检测机构平台伸缩气缸允许伸出优先条件
ORLD
LD D1196.06  ; RK_09 #2Hipot检测机构平台伸缩气缸伸出（步）
AND 815.15  ; RK_09 #2Hipot测试平台伸缩气缸伸出位标志[0015.15]
LD D1196.07  ; RK_09 #2Hipot检测机构旋转伸缩气缸伸出（步）
AND 815.12  ; RK_09 #2Hipot测试旋转伸缩气缸到位标志[0015.12]
ANDNOT H81.00  ; RK_09 #2Hipot检测机构有料记忆
ANDNOT 818.06  ; RK_09 #2Hipot测试有料感应标志[0018.06]
ANDNOT H81.01  ; RK_09 #2Hipot检测机构有OK料记忆
ANDNOT H81.02  ; RK_09 #2Hipot检测机构有NG料记忆
ANDNOT H81.03  ; RK_09 #2Hipot检测机构检测完成记忆
ORLD
AND 815.08  ; RK_09 #1Hipot测试平台伸缩气缸缩回位标志[0015.08]
LD H85.00  ; RK_10 U8_U 电池除尘上料X轴回原点记忆
ANDNOT 866.02  ; RK_10 U8_U 电池除尘上料X轴#2Hipot检测取料位标志
OR 816.03  ; RK_10 电池除尘上料机械手升降气缸上升位标志[0016.03]
ANDLD
ORLD
LD D1196.08  ; RK_09 #2Hipot检测机构旋转伸缩气缸缩回（步）
AND 815.13  ; RK_09 #2Hipot测试旋转伸缩气缸原位标志[0015.13]
AND 815.07  ; RK_09 #1Hipot测试旋转伸缩气缸原位标志[0015.07]
LD H85.00  ; RK_10 U8_U 电池除尘上料X轴回原点记忆
ANDNOT 866.02  ; RK_10 U8_U 电池除尘上料X轴#2Hipot检测取料位标志
OR 816.03  ; RK_10 电池除尘上料机械手升降气缸上升位标志[0016.03]
ANDLD
LD H40.00  ; RK_06 U8_X 电池上下料X轴回原点记忆
ANDNOT 863.07  ; RK_06 U8_X 电池上下料X轴#2Hipot检测放料位标志
LD 814.01  ; RK_06 铝壳上料升降气缸上升位标志[0014.01]
AND 814.03  ; RK_06 电池下料升降气缸上升位标志[0014.03]
ORLD
ANDLD
ORLD
LD D1196.09  ; RK_09 #2Hipot检测机构平台伸缩气缸缩回（步）
AND 815.14  ; RK_09 #2Hipot测试平台伸缩气缸缩回位标志[0015.14]
ORLD
LD D1194.01  ; RK_09 #2Hipot检测机构单步/自动循环运行中
AND W1.01  ; 自动模式
@LD D1193.15  ; RK_09 #2Hipot检测机构单步（SW）
AND D1194.10  ; RK_09 #2Hipot检测机构单步运行条件
ORLD
ANDLD
OUT D1195.01  ; RK_09 #2Hipot检测机构步进条件

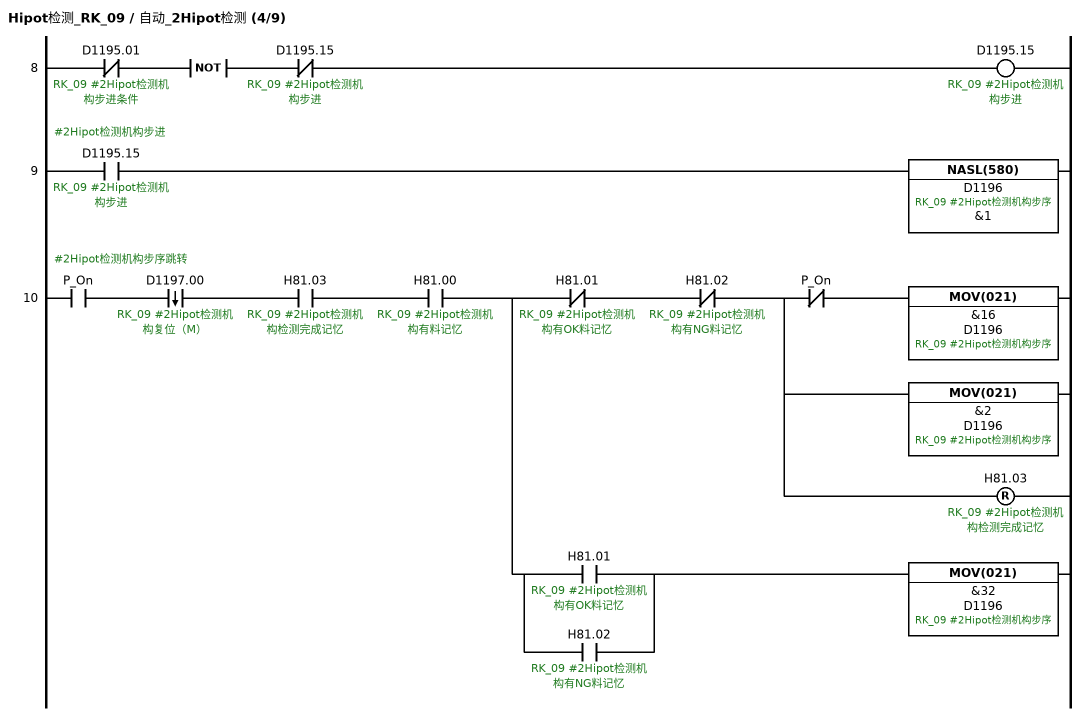
; rung 8
LDNOT D1195.01  ; RK_09 #2Hipot检测机构步进条件
NOT(520)
ANDNOT D1195.15  ; RK_09 #2Hipot检测机构步进
OUT D1195.15  ; RK_09 #2Hipot检测机构步进
; rung 9: #2Hipot检测机构步进
LD D1195.15  ; RK_09 #2Hipot检测机构步进
NASL(580) D1196 &1  ; RK_09 #2Hipot检测机构步序
; rung 10: #2Hipot检测机构步序跳转
LD P_On
%AND D1197.00  ; RK_09 #2Hipot检测机构复位（M）
AND H81.03  ; RK_09 #2Hipot检测机构检测完成记忆
AND H81.00  ; RK_09 #2Hipot检测机构有料记忆
OUT TR0
ANDNOT H81.01  ; RK_09 #2Hipot检测机构有OK料记忆
ANDNOT H81.02  ; RK_09 #2Hipot检测机构有NG料记忆
OUT TR1
ANDNOT P_On
MOV(021) &16 D1196  ; RK_09 #2Hipot检测机构步序  // RK_09 #2Hipot检测机构测试结果读取步（D1196.04）
LD TR1
MOV(021) &2 D1196  ; RK_09 #2Hipot检测机构步序  // RK_09 #2Hipot检测机构检测伸缩气缸伸出&Hipot检测数据初始化步（D1196.01）
RSET H81.03  ; RK_09 #2Hipot检测机构检测完成记忆
LD TR0
LD H81.01  ; RK_09 #2Hipot检测机构有OK料记忆
OR H81.02  ; RK_09 #2Hipot检测机构有NG料记忆
ANDLD
MOV(021) &32 D1196  ; RK_09 #2Hipot检测机构步序  // RK_09 #2Hipot检测机构检测伸缩气缸缩回步（D1196.05）

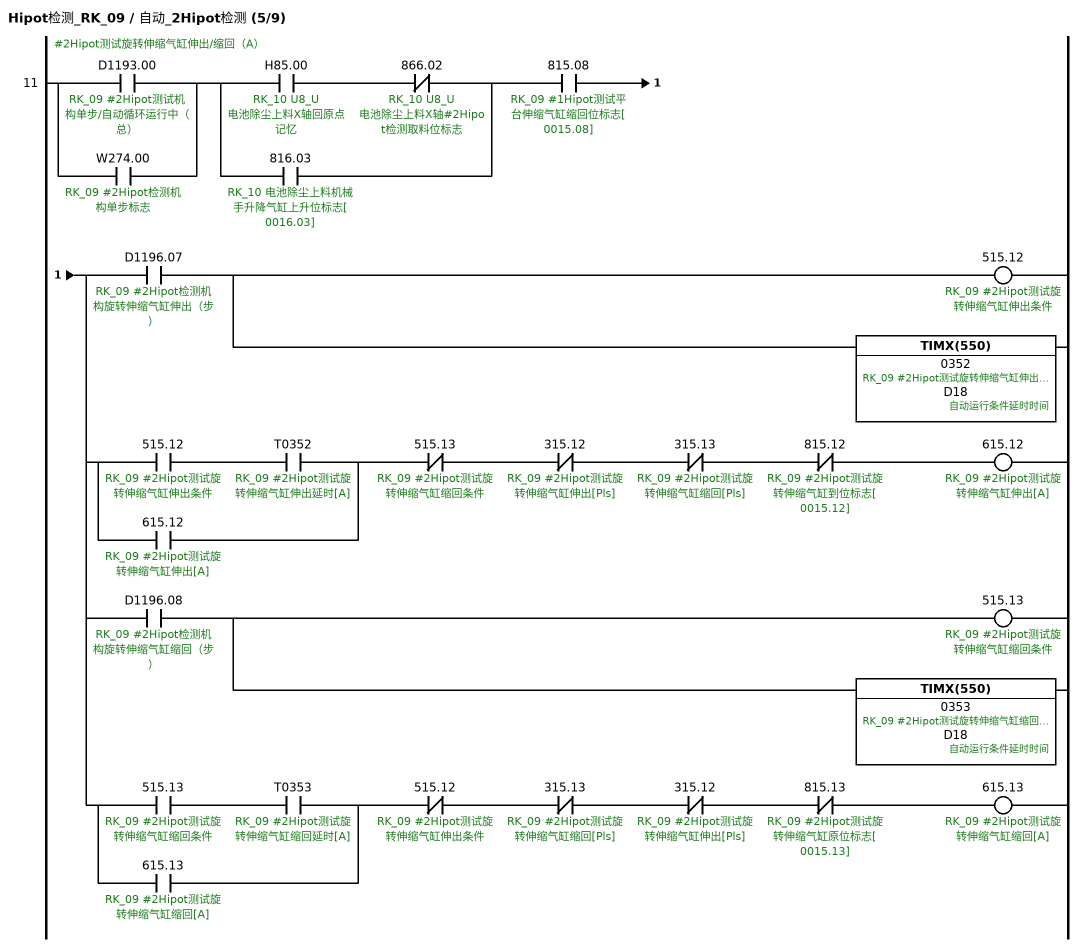
; rung 11: #2Hipot测试旋转伸缩气缸伸出/缩回（A）
LD D1193.00  ; RK_09 #2Hipot测试机构单步/自动循环运行中（总）
OR W274.00  ; RK_09 #2Hipot检测机构单步标志
LD H85.00  ; RK_10 U8_U 电池除尘上料X轴回原点记忆
ANDNOT 866.02  ; RK_10 U8_U 电池除尘上料X轴#2Hipot检测取料位标志
OR 816.03  ; RK_10 电池除尘上料机械手升降气缸上升位标志[0016.03]
ANDLD
AND 815.08  ; RK_09 #1Hipot测试平台伸缩气缸缩回位标志[0015.08]
OUT TR0
AND D1196.07  ; RK_09 #2Hipot检测机构旋转伸缩气缸伸出（步）
OUT 515.12  ; RK_09 #2Hipot测试旋转伸缩气缸伸出条件
TIMX(550) 0352 D18  ; 自动运行条件延时时间, RK_09 #2Hipot测试旋转伸缩气缸伸出延时[A]
LD TR0
LD 515.12  ; RK_09 #2Hipot测试旋转伸缩气缸伸出条件
AND T0352  ; RK_09 #2Hipot测试旋转伸缩气缸伸出延时[A]
OR 615.12  ; RK_09 #2Hipot测试旋转伸缩气缸伸出[A]
ANDLD
ANDNOT 515.13  ; RK_09 #2Hipot测试旋转伸缩气缸缩回条件
ANDNOT 315.12  ; RK_09 #2Hipot测试旋转伸缩气缸伸出[Pls]
ANDNOT 315.13  ; RK_09 #2Hipot测试旋转伸缩气缸缩回[Pls]
ANDNOT 815.12  ; RK_09 #2Hipot测试旋转伸缩气缸到位标志[0015.12]
OUT 615.12  ; RK_09 #2Hipot测试旋转伸缩气缸伸出[A]
LD TR0
AND D1196.08  ; RK_09 #2Hipot检测机构旋转伸缩气缸缩回（步）
OUT 515.13  ; RK_09 #2Hipot测试旋转伸缩气缸缩回条件
TIMX(550) 0353 D18  ; 自动运行条件延时时间, RK_09 #2Hipot测试旋转伸缩气缸缩回延时[A]
LD TR0
LD 515.13  ; RK_09 #2Hipot测试旋转伸缩气缸缩回条件
AND T0353  ; RK_09 #2Hipot测试旋转伸缩气缸缩回延时[A]
OR 615.13  ; RK_09 #2Hipot测试旋转伸缩气缸缩回[A]
ANDLD
ANDNOT 515.12  ; RK_09 #2Hipot测试旋转伸缩气缸伸出条件
ANDNOT 315.13  ; RK_09 #2Hipot测试旋转伸缩气缸缩回[Pls]
ANDNOT 315.12  ; RK_09 #2Hipot测试旋转伸缩气缸伸出[Pls]
ANDNOT 815.13  ; RK_09 #2Hipot测试旋转伸缩气缸原位标志[0015.13]
OUT 615.13  ; RK_09 #2Hipot测试旋转伸缩气缸缩回[A]

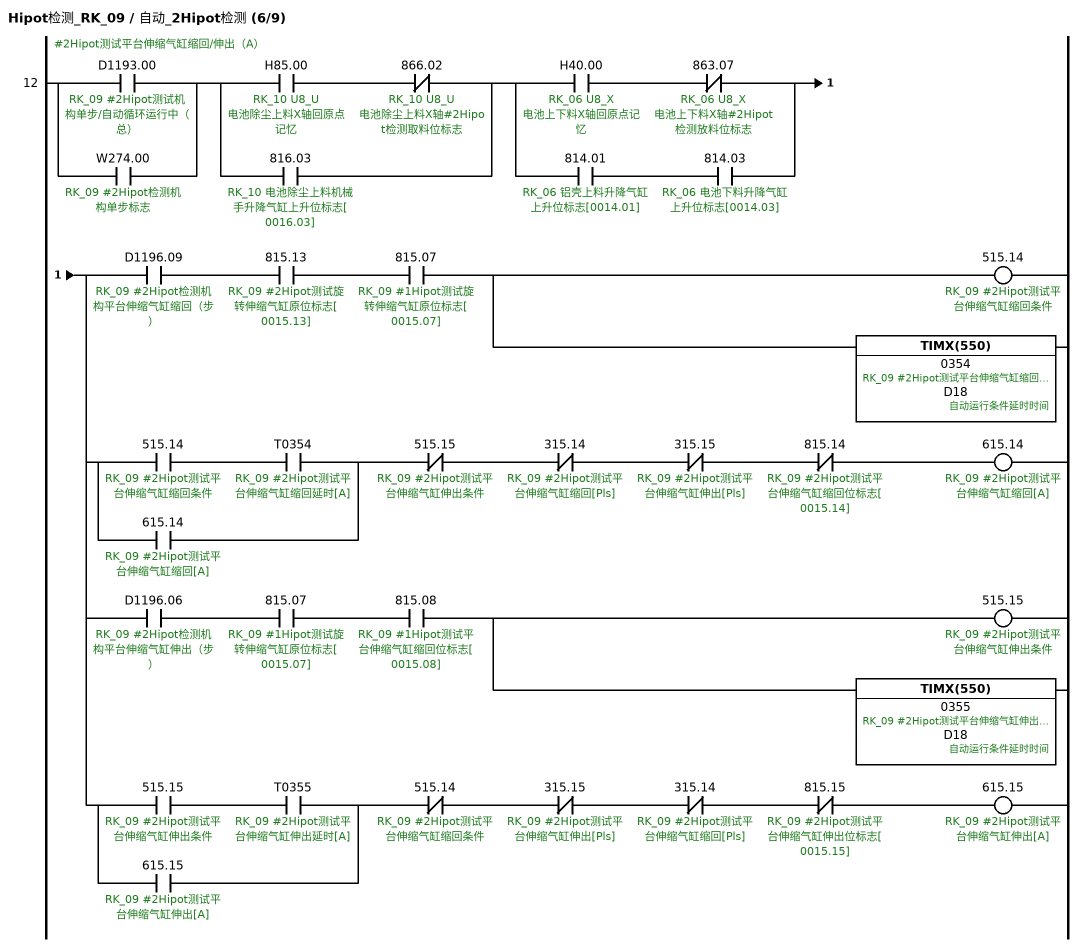
; rung 12: #2Hipot测试平台伸缩气缸缩回/伸出（A）
LD D1193.00  ; RK_09 #2Hipot测试机构单步/自动循环运行中（总）
OR W274.00  ; RK_09 #2Hipot检测机构单步标志
LD H85.00  ; RK_10 U8_U 电池除尘上料X轴回原点记忆
ANDNOT 866.02  ; RK_10 U8_U 电池除尘上料X轴#2Hipot检测取料位标志
OR 816.03  ; RK_10 电池除尘上料机械手升降气缸上升位标志[0016.03]
ANDLD
LD H40.00  ; RK_06 U8_X 电池上下料X轴回原点记忆
ANDNOT 863.07  ; RK_06 U8_X 电池上下料X轴#2Hipot检测放料位标志
LD 814.01  ; RK_06 铝壳上料升降气缸上升位标志[0014.01]
AND 814.03  ; RK_06 电池下料升降气缸上升位标志[0014.03]
ORLD
ANDLD
OUT TR0
AND D1196.09  ; RK_09 #2Hipot检测机构平台伸缩气缸缩回（步）
AND 815.13  ; RK_09 #2Hipot测试旋转伸缩气缸原位标志[0015.13]
AND 815.07  ; RK_09 #1Hipot测试旋转伸缩气缸原位标志[0015.07]
OUT 515.14  ; RK_09 #2Hipot测试平台伸缩气缸缩回条件
TIMX(550) 0354 D18  ; 自动运行条件延时时间, RK_09 #2Hipot测试平台伸缩气缸缩回延时[A]
LD TR0
LD 515.14  ; RK_09 #2Hipot测试平台伸缩气缸缩回条件
AND T0354  ; RK_09 #2Hipot测试平台伸缩气缸缩回延时[A]
OR 615.14  ; RK_09 #2Hipot测试平台伸缩气缸缩回[A]
ANDLD
ANDNOT 515.15  ; RK_09 #2Hipot测试平台伸缩气缸伸出条件
ANDNOT 315.14  ; RK_09 #2Hipot测试平台伸缩气缸缩回[Pls]
ANDNOT 315.15  ; RK_09 #2Hipot测试平台伸缩气缸伸出[Pls]
ANDNOT 815.14  ; RK_09 #2Hipot测试平台伸缩气缸缩回位标志[0015.14]
OUT 615.14  ; RK_09 #2Hipot测试平台伸缩气缸缩回[A]
LD TR0
AND D1196.06  ; RK_09 #2Hipot检测机构平台伸缩气缸伸出（步）
AND 815.07  ; RK_09 #1Hipot测试旋转伸缩气缸原位标志[0015.07]
AND 815.08  ; RK_09 #1Hipot测试平台伸缩气缸缩回位标志[0015.08]
OUT 515.15  ; RK_09 #2Hipot测试平台伸缩气缸伸出条件
TIMX(550) 0355 D18  ; 自动运行条件延时时间, RK_09 #2Hipot测试平台伸缩气缸伸出延时[A]
LD TR0
LD 515.15  ; RK_09 #2Hipot测试平台伸缩气缸伸出条件
AND T0355  ; RK_09 #2Hipot测试平台伸缩气缸伸出延时[A]
OR 615.15  ; RK_09 #2Hipot测试平台伸缩气缸伸出[A]
ANDLD
ANDNOT 515.14  ; RK_09 #2Hipot测试平台伸缩气缸缩回条件
ANDNOT 315.15  ; RK_09 #2Hipot测试平台伸缩气缸伸出[Pls]
ANDNOT 315.14  ; RK_09 #2Hipot测试平台伸缩气缸缩回[Pls]
ANDNOT 815.15  ; RK_09 #2Hipot测试平台伸缩气缸伸出位标志[0015.15]
OUT 615.15  ; RK_09 #2Hipot测试平台伸缩气缸伸出[A]

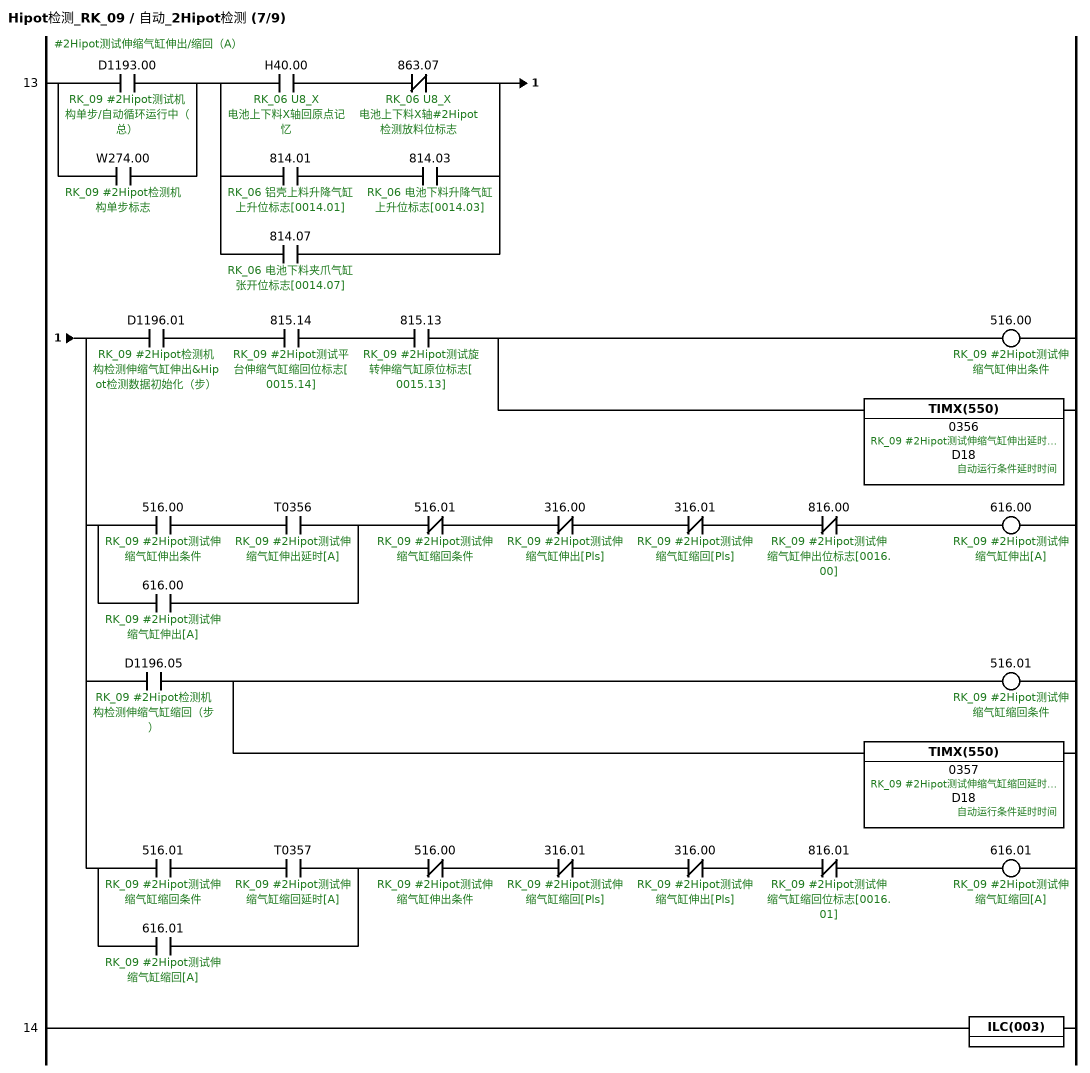
; rung 13: #2Hipot测试伸缩气缸伸出/缩回（A）
LD D1193.00  ; RK_09 #2Hipot测试机构单步/自动循环运行中（总）
OR W274.00  ; RK_09 #2Hipot检测机构单步标志
LD H40.00  ; RK_06 U8_X 电池上下料X轴回原点记忆
ANDNOT 863.07  ; RK_06 U8_X 电池上下料X轴#2Hipot检测放料位标志
LD 814.01  ; RK_06 铝壳上料升降气缸上升位标志[0014.01]
AND 814.03  ; RK_06 电池下料升降气缸上升位标志[0014.03]
ORLD
OR 814.07  ; RK_06 电池下料夹爪气缸张开位标志[0014.07]
ANDLD
OUT TR0
AND D1196.01  ; RK_09 #2Hipot检测机构检测伸缩气缸伸出&Hipot检测数据初始化（步）
AND 815.14  ; RK_09 #2Hipot测试平台伸缩气缸缩回位标志[0015.14]
AND 815.13  ; RK_09 #2Hipot测试旋转伸缩气缸原位标志[0015.13]
OUT 516.00  ; RK_09 #2Hipot测试伸缩气缸伸出条件
TIMX(550) 0356 D18  ; 自动运行条件延时时间, RK_09 #2Hipot测试伸缩气缸伸出延时[A]
LD TR0
LD 516.00  ; RK_09 #2Hipot测试伸缩气缸伸出条件
AND T0356  ; RK_09 #2Hipot测试伸缩气缸伸出延时[A]
OR 616.00  ; RK_09 #2Hipot测试伸缩气缸伸出[A]
ANDLD
ANDNOT 516.01  ; RK_09 #2Hipot测试伸缩气缸缩回条件
ANDNOT 316.00  ; RK_09 #2Hipot测试伸缩气缸伸出[Pls]
ANDNOT 316.01  ; RK_09 #2Hipot测试伸缩气缸缩回[Pls]
ANDNOT 816.00  ; RK_09 #2Hipot测试伸缩气缸伸出位标志[0016.00]
OUT 616.00  ; RK_09 #2Hipot测试伸缩气缸伸出[A]
LD TR0
AND D1196.05  ; RK_09 #2Hipot检测机构检测伸缩气缸缩回（步）
OUT 516.01  ; RK_09 #2Hipot测试伸缩气缸缩回条件
TIMX(550) 0357 D18  ; 自动运行条件延时时间, RK_09 #2Hipot测试伸缩气缸缩回延时[A]
LD TR0
LD 516.01  ; RK_09 #2Hipot测试伸缩气缸缩回条件
AND T0357  ; RK_09 #2Hipot测试伸缩气缸缩回延时[A]
OR 616.01  ; RK_09 #2Hipot测试伸缩气缸缩回[A]
ANDLD
ANDNOT 516.00  ; RK_09 #2Hipot测试伸缩气缸伸出条件
ANDNOT 316.01  ; RK_09 #2Hipot测试伸缩气缸缩回[Pls]
ANDNOT 316.00  ; RK_09 #2Hipot测试伸缩气缸伸出[Pls]
ANDNOT 816.01  ; RK_09 #2Hipot测试伸缩气缸缩回位标志[0016.01]
OUT 616.01  ; RK_09 #2Hipot测试伸缩气缸缩回[A]
; rung 14
ILC(003)

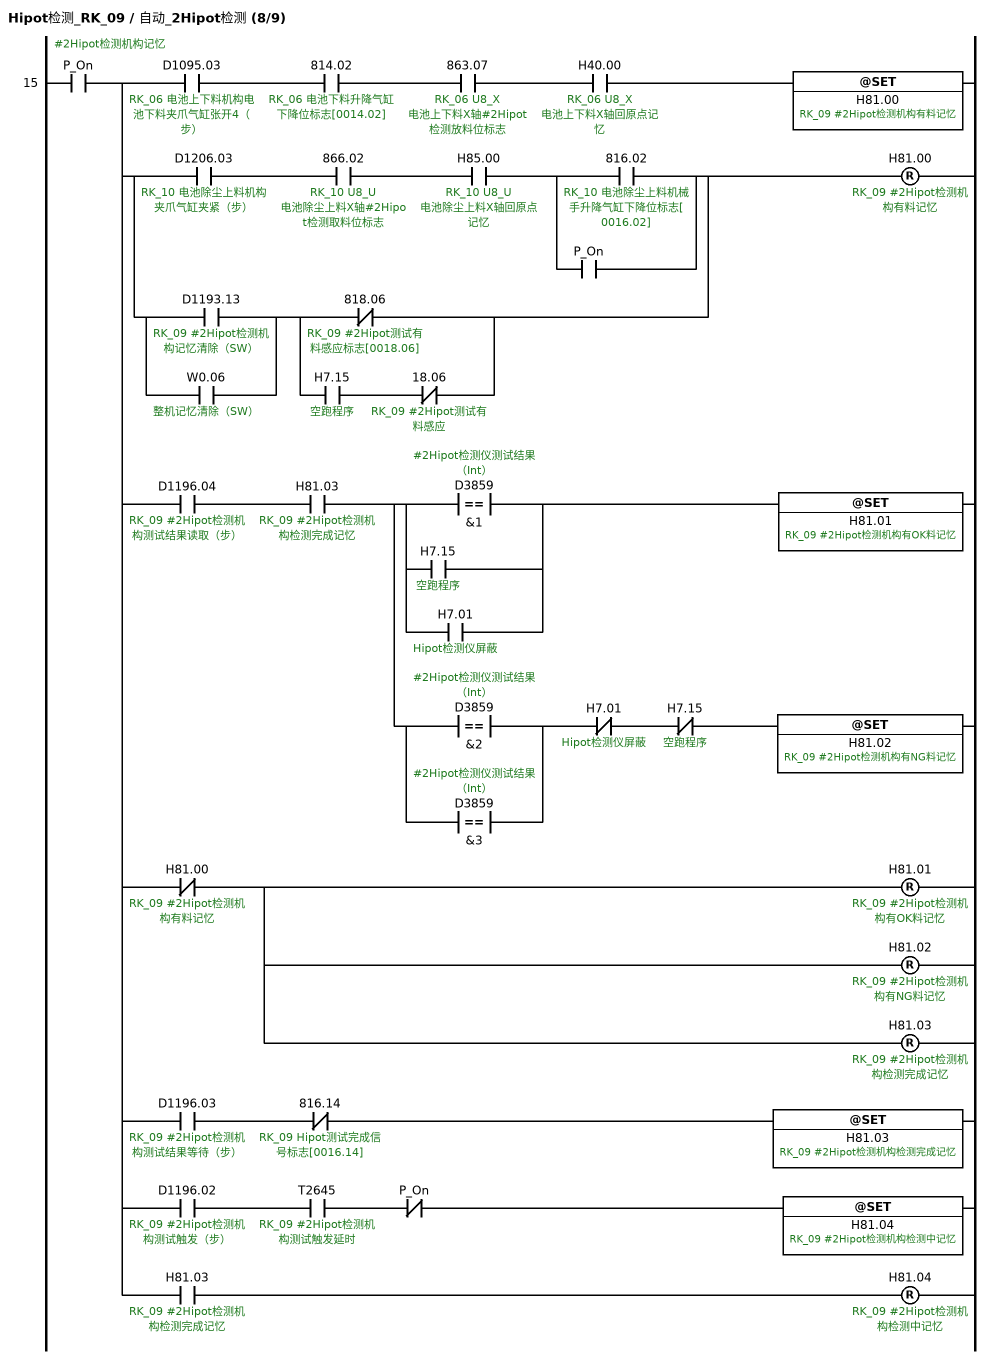
; rung 15: #2Hipot检测机构记忆
LD P_On
OUT TR0
AND D1095.03  ; RK_06 电池上下料机构电池下料夹爪气缸张开4（步）
AND 814.02  ; RK_06 电池下料升降气缸下降位标志[0014.02]
AND 863.07  ; RK_06 U8_X 电池上下料X轴#2Hipot检测放料位标志
AND H40.00  ; RK_06 U8_X 电池上下料X轴回原点记忆
@SET H81.00  ; RK_09 #2Hipot检测机构有料记忆
LD TR0
LD D1206.03  ; RK_10 电池除尘上料机构夹爪气缸夹紧（步）
AND 866.02  ; RK_10 U8_U 电池除尘上料X轴#2Hipot检测取料位标志
AND H85.00  ; RK_10 U8_U 电池除尘上料X轴回原点记忆
LD 816.02  ; RK_10 电池除尘上料机械手升降气缸下降位标志[0016.02]
OR P_On
ANDLD
LD D1193.13  ; RK_09 #2Hipot检测机构记忆清除（SW）
OR W0.06  ; 整机记忆清除（SW）
LDNOT 818.06  ; RK_09 #2Hipot测试有料感应标志[0018.06]
LD H7.15  ; 空跑程序
ANDNOT 18.06  ; RK_09 #2Hipot测试有料感应
ORLD
ANDLD
ORLD
ANDLD
RSET H81.00  ; RK_09 #2Hipot检测机构有料记忆
LD TR0
AND D1196.04  ; RK_09 #2Hipot检测机构测试结果读取（步）
AND H81.03  ; RK_09 #2Hipot检测机构检测完成记忆
OUT TR1
LD=(300) D3859 &1  ; #2Hipot检测仪测试结果（Int）
OR H7.15  ; 空跑程序
OR H7.01  ; Hipot检测仪屏蔽
ANDLD
@SET H81.01  ; RK_09 #2Hipot检测机构有OK料记忆
LD TR1
LD=(300) D3859 &2  ; #2Hipot检测仪测试结果（Int）
OR=(300) D3859 &3  ; #2Hipot检测仪测试结果（Int）
ANDLD
ANDNOT H7.01  ; Hipot检测仪屏蔽
ANDNOT H7.15  ; 空跑程序
@SET H81.02  ; RK_09 #2Hipot检测机构有NG料记忆
LD TR0
ANDNOT H81.00  ; RK_09 #2Hipot检测机构有料记忆
RSET H81.01  ; RK_09 #2Hipot检测机构有OK料记忆
RSET H81.02  ; RK_09 #2Hipot检测机构有NG料记忆
RSET H81.03  ; RK_09 #2Hipot检测机构检测完成记忆
LD TR0
AND D1196.03  ; RK_09 #2Hipot检测机构测试结果等待（步）
ANDNOT 816.14  ; RK_09 Hipot测试完成信号标志[0016.14]
@SET H81.03  ; RK_09 #2Hipot检测机构检测完成记忆
LD TR0
AND D1196.02  ; RK_09 #2Hipot检测机构测试触发（步）
AND T2645  ; RK_09 #2Hipot检测机构测试触发延时
ANDNOT P_On
@SET H81.04  ; RK_09 #2Hipot检测机构检测中记忆
LD TR0
AND H81.03  ; RK_09 #2Hipot检测机构检测完成记忆
RSET H81.04  ; RK_09 #2Hipot检测机构检测中记忆

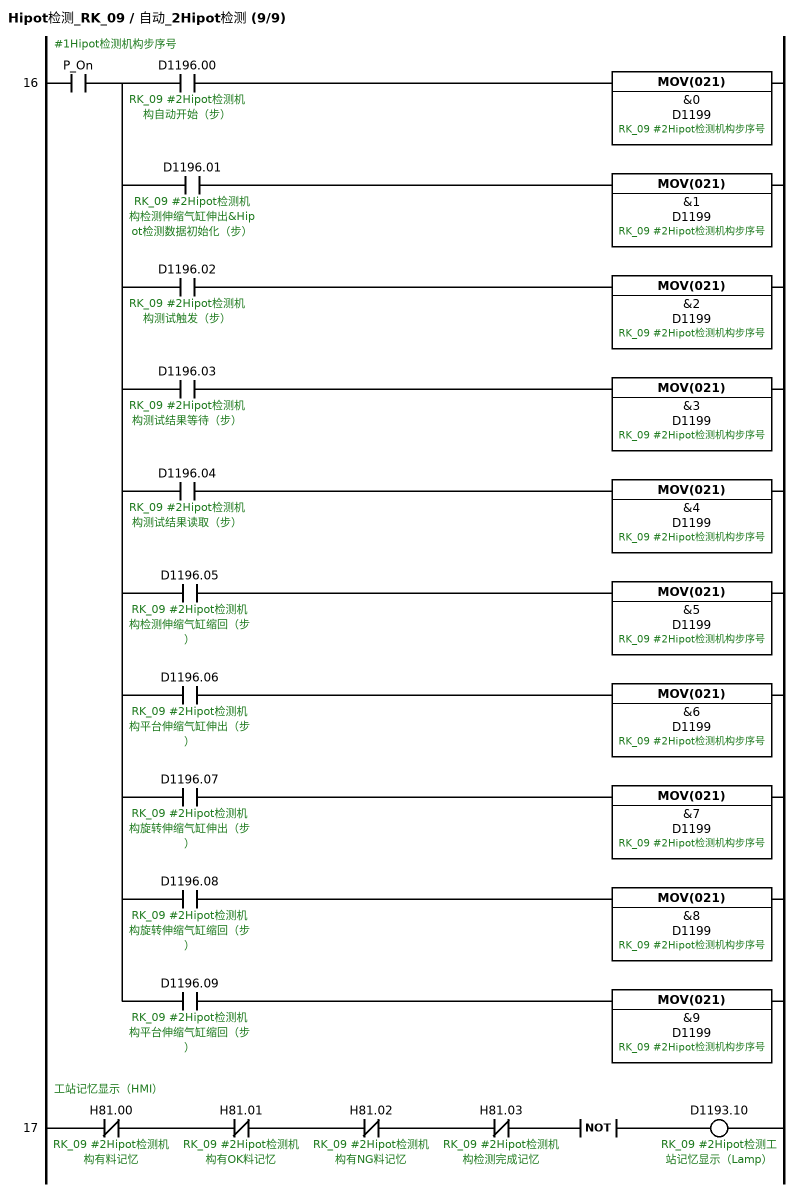
; rung 16: #1Hipot检测机构步序号
LD P_On
OUT TR0
AND D1196.00  ; RK_09 #2Hipot检测机构自动开始（步）
MOV(021) &0 D1199  ; RK_09 #2Hipot检测机构步序号
LD TR0
AND D1196.01  ; RK_09 #2Hipot检测机构检测伸缩气缸伸出&Hipot检测数据初始化（步）
MOV(021) &1 D1199  ; RK_09 #2Hipot检测机构步序号
LD TR0
AND D1196.02  ; RK_09 #2Hipot检测机构测试触发（步）
MOV(021) &2 D1199  ; RK_09 #2Hipot检测机构步序号
LD TR0
AND D1196.03  ; RK_09 #2Hipot检测机构测试结果等待（步）
MOV(021) &3 D1199  ; RK_09 #2Hipot检测机构步序号
LD TR0
AND D1196.04  ; RK_09 #2Hipot检测机构测试结果读取（步）
MOV(021) &4 D1199  ; RK_09 #2Hipot检测机构步序号
LD TR0
AND D1196.05  ; RK_09 #2Hipot检测机构检测伸缩气缸缩回（步）
MOV(021) &5 D1199  ; RK_09 #2Hipot检测机构步序号
LD TR0
AND D1196.06  ; RK_09 #2Hipot检测机构平台伸缩气缸伸出（步）
MOV(021) &6 D1199  ; RK_09 #2Hipot检测机构步序号
LD TR0
AND D1196.07  ; RK_09 #2Hipot检测机构旋转伸缩气缸伸出（步）
MOV(021) &7 D1199  ; RK_09 #2Hipot检测机构步序号
LD TR0
AND D1196.08  ; RK_09 #2Hipot检测机构旋转伸缩气缸缩回（步）
MOV(021) &8 D1199  ; RK_09 #2Hipot检测机构步序号
LD TR0
AND D1196.09  ; RK_09 #2Hipot检测机构平台伸缩气缸缩回（步）
MOV(021) &9 D1199  ; RK_09 #2Hipot检测机构步序号
; rung 17: 工站记忆显示（HMI）
LDNOT H81.00  ; RK_09 #2Hipot检测机构有料记忆
ANDNOT H81.01  ; RK_09 #2Hipot检测机构有OK料记忆
ANDNOT H81.02  ; RK_09 #2Hipot检测机构有NG料记忆
ANDNOT H81.03  ; RK_09 #2Hipot检测机构检测完成记忆
NOT(520)
OUT D1193.10  ; RK_09 #2Hipot检测工站记忆显示（Lamp）

### Section 复位

